   1:  PR[91,1] = PR[90,1] + 40.590;
   1:  PR[91,2] = PR[90,2] + 10.194;
   1:L PR[91] R[100]mm/sec CNT100;
   1:  PR[91,1] = PR[90,1] + 38.016;
   1:  PR[91,2] = PR[90,2] + 13.467;
   1:L PR[91] R[100]mm/sec CNT100;
   1:  PR[91,1] = PR[90,1] + 37.291;
   1:  PR[91,2] = PR[90,2] + 14.026;
   1:L PR[91] R[100]mm/sec CNT100;
   1:  PR[91,1] = PR[90,1] + 33.908;
   1:  PR[91,2] = PR[90,2] + 16.575;
   1:L PR[91] R[100]mm/sec CNT100;
   1:  PR[91,1] = PR[90,1] + 29.117;
   1:  PR[91,2] = PR[90,2] + 18.537;
   1:L PR[91] R[100]mm/sec CNT100;
   1:  PR[91,1] = PR[90,1] + 28.399;
   1:  PR[91,2] = PR[90,2] + 18.634;
   1:L PR[91] R[100]mm/sec CNT100;
   1:  PR[91,1] = PR[90,1] + 23.987;
   1:  PR[91,2] = PR[90,2] + 19.202;
   1:L PR[91] R[100]mm/sec CNT100;
   1:  PR[91,1] = PR[90,1] + 18.842;
   1:  PR[91,2] = PR[90,2] + 18.522;
   1:L PR[91] R[100]mm/sec CNT100;
   1:  PR[91,1] = PR[90,1] + 14.039;
   1:  PR[91,2] = PR[90,2] + 16.538;
   1:L PR[91] R[100]mm/sec CNT100;
   1:  PR[91,1] = PR[90,1] + 9.906;
   1:  PR[91,2] = PR[90,2] + 13.378;
   1:L PR[91] R[100]mm/sec CNT100;
   1:  PR[91,1] = PR[90,1] + 6.730;
   1:  PR[91,2] = PR[90,2] + 9.250;
   1:L PR[91] R[100]mm/sec CNT100;
   1:  PR[91,1] = PR[90,1] + 4.730;
   1:  PR[91,2] = PR[90,2] + 4.439;
   1:L PR[91] R[100]mm/sec CNT100;
   1:  PR[91,1] = PR[90,1] + 4.049;
   1:  PR[91,2] = PR[90,2] + -0.729;
   1:L PR[91] R[100]mm/sec CNT100;
   1:  PR[91,1] = PR[90,1] + 4.732;
   1:  PR[91,2] = PR[90,2] + -5.902;
   1:L PR[91] R[100]mm/sec CNT100;
   1:  PR[91,1] = PR[90,1] + 6.735;
   1:  PR[91,2] = PR[90,2] + -10.718;
   1:L PR[91] R[100]mm/sec CNT100;
   1:  PR[91,1] = PR[90,1] + 9.916;
   1:  PR[91,2] = PR[90,2] + -14.847;
   1:L PR[91] R[100]mm/sec CNT100;
   1:  PR[91,1] = PR[90,1] + 14.056;
   1:  PR[91,2] = PR[90,2] + -18.006;
   1:L PR[91] R[100]mm/sec CNT100;
   1:  PR[91,1] = PR[90,1] + 18.865;
   1:  PR[91,2] = PR[90,2] + -19.987;
   1:L PR[91] R[100]mm/sec CNT100;
   1:  PR[91,1] = PR[90,1] + 24.014;
   1:  PR[91,2] = PR[90,2] + -20.661;
   1:L PR[91] R[100]mm/sec CNT100;
   1:  PR[91,1] = PR[90,1] + 28.429;
   1:  PR[91,2] = PR[90,2] + -20.085;
   1:L PR[91] R[100]mm/sec CNT100;
   1:  PR[91,1] = PR[90,1] + 29.148;
   1:  PR[91,2] = PR[90,2] + -19.987;
   1:L PR[91] R[100]mm/sec CNT100;
   1:  PR[91,1] = PR[90,1] + 33.936;
   1:  PR[91,2] = PR[90,2] + -18.017;
   1:L PR[91] R[100]mm/sec CNT100;
   1:  PR[91,1] = PR[90,1] + 38.048;
   1:  PR[91,2] = PR[90,2] + -14.892;
   1:L PR[91] R[100]mm/sec CNT100;
   1:  PR[91,1] = PR[90,1] + 40.630;
   1:  PR[91,2] = PR[90,2] + -11.589;
   1:L PR[91] R[100]mm/sec CNT100;
   1:  PR[91,1] = PR[90,1] + 41.273;
   1:  PR[91,2] = PR[90,2] + -10.747;
   1:L PR[91] R[100]mm/sec CNT100;
   1:  PR[91,1] = PR[90,1] + 41.543;
   1:  PR[91,2] = PR[90,2] + -10.255;
   1:L PR[91] R[100]mm/sec CNT100;
   1:  PR[91,1] = PR[90,1] + 41.867;
   1:  PR[91,2] = PR[90,2] + -9.470;
   1:L PR[91] R[100]mm/sec CNT100;
   1:  PR[91,1] = PR[90,1] + 44.364;
   1:  PR[91,2] = PR[90,2] + -3.909;
   1:L PR[91] R[100]mm/sec CNT100;
   1:  PR[91,1] = PR[90,1] + 47.704;
   1:  PR[91,2] = PR[90,2] + -10.331;
   1:L PR[91] R[100]mm/sec CNT100;
   1:  PR[91,1] = PR[90,1] + 48.926;
   1:  PR[91,2] = PR[90,2] + -11.795;
   1:L PR[91] R[100]mm/sec CNT100;
   1:  PR[91,1] = PR[90,1] + 51.775;
   1:  PR[91,2] = PR[90,2] + -14.772;
   1:L PR[91] R[100]mm/sec CNT100;
   1:  PR[91,1] = PR[90,1] + 52.056;
   1:  PR[91,2] = PR[90,2] + -14.978;
   1:L PR[91] R[100]mm/sec CNT100;
   1:  PR[91,1] = PR[90,1] + 53.337;
   1:  PR[91,2] = PR[90,2] + -15.767;
   1:L PR[91] R[100]mm/sec CNT100;
   1:  PR[91,1] = PR[90,1] + 56.402;
   1:  PR[91,2] = PR[90,2] + -17.898;
   1:L PR[91] R[100]mm/sec CNT100;
   1:  PR[91,1] = PR[90,1] + 57.333;
   1:  PR[91,2] = PR[90,2] + -18.350;
   1:L PR[91] R[100]mm/sec CNT100;
   1:  PR[91,1] = PR[90,1] + 60.886;
   1:  PR[91,2] = PR[90,2] + -19.737;
   1:L PR[91] R[100]mm/sec CNT100;
   1:  PR[91,1] = PR[90,1] + 63.586;
   1:  PR[91,2] = PR[90,2] + -20.396;
   1:L PR[91] R[100]mm/sec CNT100;
   1:  PR[91,1] = PR[90,1] + 65.452;
   1:  PR[91,2] = PR[90,2] + -20.674;
   1:L PR[91] R[100]mm/sec CNT100;
   1:  PR[91,1] = PR[90,1] + 69.656;
   1:  PR[91,2] = PR[90,2] + -20.825;
   1:L PR[91] R[100]mm/sec CNT100;
   1:  PR[91,1] = PR[90,1] + 69.952;
   1:  PR[91,2] = PR[90,2] + -20.804;
   1:L PR[91] R[100]mm/sec CNT100;
   1:  PR[91,1] = PR[90,1] + 71.659;
   1:  PR[91,2] = PR[90,2] + -20.520;
   1:L PR[91] R[100]mm/sec CNT100;
   1:  PR[91,1] = PR[90,1] + 74.623;
   1:  PR[91,2] = PR[90,2] + -20.055;
   1:L PR[91] R[100]mm/sec CNT100;
   1:  PR[91,1] = PR[90,1] + 75.033;
   1:  PR[91,2] = PR[90,2] + -19.903;
   1:L PR[91] R[100]mm/sec CNT100;
   1:  PR[91,1] = PR[90,1] + 78.943;
   1:  PR[91,2] = PR[90,2] + -18.404;
   1:L PR[91] R[100]mm/sec CNT100;
   1:  PR[91,1] = PR[90,1] + 80.020;
   1:  PR[91,2] = PR[90,2] + -17.717;
   1:L PR[91] R[100]mm/sec CNT100;
   1:  PR[91,1] = PR[90,1] + 82.749;
   1:  PR[91,2] = PR[90,2] + -15.933;
   1:L PR[91] R[100]mm/sec CNT100;
   1:  PR[91,1] = PR[90,1] + 84.089;
   1:  PR[91,2] = PR[90,2] + -14.597;
   1:L PR[91] R[100]mm/sec CNT100;
   1:  PR[91,1] = PR[90,1] + 85.881;
   1:  PR[91,2] = PR[90,2] + -12.773;
   1:L PR[91] R[100]mm/sec CNT100;
   1:  PR[91,1] = PR[90,1] + 88.217;
   1:  PR[91,2] = PR[90,2] + -9.066;
   1:L PR[91] R[100]mm/sec CNT100;
   1:  PR[91,1] = PR[90,1] + 89.654;
   1:  PR[91,2] = PR[90,2] + -4.990;
   1:L PR[91] R[100]mm/sec CNT100;
   1:  PR[91,1] = PR[90,1] + 90.143;
   1:  PR[91,2] = PR[90,2] + -0.729;
   1:L PR[91] R[100]mm/sec CNT100;
   1:  PR[91,1] = PR[90,1] + 89.654;
   1:  PR[91,2] = PR[90,2] + 3.531;
   1:L PR[91] R[100]mm/sec CNT100;
   1:  PR[91,1] = PR[90,1] + 88.218;
   1:  PR[91,2] = PR[90,2] + 7.603;
   1:L PR[91] R[100]mm/sec CNT100;
   1:  PR[91,1] = PR[90,1] + 86.960;
   1:  PR[91,2] = PR[90,2] + 9.583;
   1:L PR[91] R[100]mm/sec CNT100;
   1:  PR[91,1] = PR[90,1] + 85.883;
   1:  PR[91,2] = PR[90,2] + 11.309;
   1:L PR[91] R[100]mm/sec CNT100;
   1:  PR[91,1] = PR[90,1] + 84.452;
   1:  PR[91,2] = PR[90,2] + 12.734;
   1:L PR[91] R[100]mm/sec CNT100;
   1:  PR[91,1] = PR[90,1] + 82.749;
   1:  PR[91,2] = PR[90,2] + 14.471;
   1:L PR[91] R[100]mm/sec CNT100;
   1:  PR[91,1] = PR[90,1] + 81.417;
   1:  PR[91,2] = PR[90,2] + 15.317;
   1:L PR[91] R[100]mm/sec CNT100;
   1:  PR[91,1] = PR[90,1] + 78.943;
   1:  PR[91,2] = PR[90,2] + 16.942;
   1:L PR[91] R[100]mm/sec CNT100;
   1:  PR[91,1] = PR[90,1] + 77.998;
   1:  PR[91,2] = PR[90,2] + 17.288;
   1:L PR[91] R[100]mm/sec CNT100;
   1:  PR[91,1] = PR[90,1] + 74.607;
   1:  PR[91,2] = PR[90,2] + 18.598;
   1:L PR[91] R[100]mm/sec CNT100;
   1:  PR[91,1] = PR[90,1] + 71.659;
   1:  PR[91,2] = PR[90,2] + 19.061;
   1:L PR[91] R[100]mm/sec CNT100;
   1:  PR[91,1] = PR[90,1] + 69.952;
   1:  PR[91,2] = PR[90,2] + 19.345;
   1:L PR[91] R[100]mm/sec CNT100TB   .50sec,CALL END_PUD;
   1:  PR[92] = PR[91];
   1:  PR[92,3] = PR[92,3] + 20;
   1:J PR[92] 10% FINE;
   1:  PR[91,1] = PR[90,1] + -21.225;
   1:  PR[91,2] = PR[90,2] + -20.035;
   1:  PR[92] = PR[91];
   1:  PR[92,3] = PR[92,3] + 20;
   1:J PR[92] 10% FINE;
   1:L PR[91] R[100]mm/sec CNT100;
   1:  CALL LASER_DRAHT_START;
   1:  PR[91,1] = PR[90,1] + -17.834;
   1:  PR[91,2] = PR[90,2] + -19.755;
   1:L PR[91] R[100]mm/sec CNT100;
   1:  PR[91,1] = PR[90,1] + -16.393;
   1:  PR[91,2] = PR[90,2] + -19.403;
   1:L PR[91] R[100]mm/sec CNT100;
   1:  PR[91,1] = PR[90,1] + -13.614;
   1:  PR[91,2] = PR[90,2] + -18.541;
   1:L PR[91] R[100]mm/sec CNT100;
   1:  PR[91,1] = PR[90,1] + -11.836;
   1:  PR[91,2] = PR[90,2] + -17.662;
   1:L PR[91] R[100]mm/sec CNT100;
   1:  PR[91,1] = PR[90,1] + -9.749;
   1:  PR[91,2] = PR[90,2] + -16.459;
   1:L PR[91] R[100]mm/sec CNT100;
   1:  PR[91,1] = PR[90,1] + -7.849;
   1:  PR[91,2] = PR[90,2] + -14.914;
   1:L PR[91] R[100]mm/sec CNT100;
   1:  PR[91,1] = PR[90,1] + -6.429;
   1:  PR[91,2] = PR[90,2] + -13.596;
   1:L PR[91] R[100]mm/sec CNT100;
   1:  PR[91,1] = PR[90,1] + -4.688;
   1:  PR[91,2] = PR[90,2] + -11.349;
   1:L PR[91] R[100]mm/sec CNT100;
   1:  PR[91,1] = PR[90,1] + -3.827;
   1:  PR[91,2] = PR[90,2] + -10.067;
   1:L PR[91] R[100]mm/sec CNT100;
   1:  PR[91,1] = PR[90,1] + -2.535;
   1:  PR[91,2] = PR[90,2] + -7.218;
   1:L PR[91] R[100]mm/sec CNT100;
   1:  PR[91,1] = PR[90,1] + -2.094;
   1:  PR[91,2] = PR[90,2] + -6.035;
   1:L PR[91] R[100]mm/sec CNT100;
   1:  PR[91,1] = PR[90,1] + -1.483;
   1:  PR[91,2] = PR[90,2] + -2.786;
   1:L PR[91] R[100]mm/sec CNT100;
   1:  PR[91,1] = PR[90,1] + -1.346;
   1:  PR[91,2] = PR[90,2] + -1.651;
   1:L PR[91] R[100]mm/sec CNT100;
   1:  PR[91,1] = PR[90,1] + -1.323;
   1:  PR[91,2] = PR[90,2] + -0.821;
   1:L PR[91] R[100]mm/sec CNT100;
   1:  PR[91,1] = PR[90,1] + -1.464;
   1:  PR[91,2] = PR[90,2] + 0.357;
   1:L PR[91] R[100]mm/sec CNT100;
   1:  PR[91,1] = PR[90,1] + -1.499;
   1:  PR[91,2] = PR[90,2] + 1.403;
   1:L PR[91] R[100]mm/sec CNT100;
   1:  PR[91,1] = PR[90,1] + -2.091;
   1:  PR[91,2] = PR[90,2] + 4.565;
   1:L PR[91] R[100]mm/sec CNT100;
   1:  PR[91,1] = PR[90,1] + -2.532;
   1:  PR[91,2] = PR[90,2] + 5.748;
   1:L PR[91] R[100]mm/sec CNT100;
   1:  PR[91,1] = PR[90,1] + -3.821;
   1:  PR[91,2] = PR[90,2] + 8.599;
   1:L PR[91] R[100]mm/sec CNT100;
   1:  PR[91,1] = PR[90,1] + -4.683;
   1:  PR[91,2] = PR[90,2] + 9.880;
   1:L PR[91] R[100]mm/sec CNT100;
   1:  PR[91,1] = PR[90,1] + -6.422;
   1:  PR[91,2] = PR[90,2] + 12.130;
   1:L PR[91] R[100]mm/sec CNT100;
   1:  PR[91,1] = PR[90,1] + -7.842;
   1:  PR[91,2] = PR[90,2] + 13.448;
   1:L PR[91] R[100]mm/sec CNT100;
   1:  PR[91,1] = PR[90,1] + -9.742;
   1:  PR[91,2] = PR[90,2] + 14.996;
   1:L PR[91] R[100]mm/sec CNT100;
   1:  PR[91,1] = PR[90,1] + -11.830;
   1:  PR[91,2] = PR[90,2] + 16.199;
   1:L PR[91] R[100]mm/sec CNT100;
   1:  PR[91,1] = PR[90,1] + -13.608;
   1:  PR[91,2] = PR[90,2] + 17.080;
   1:L PR[91] R[100]mm/sec CNT100;
   1:  PR[91,1] = PR[90,1] + -16.388;
   1:  PR[91,2] = PR[90,2] + 17.942;
   1:L PR[91] R[100]mm/sec CNT100;
   1:  PR[91,1] = PR[90,1] + -17.830;
   1:  PR[91,2] = PR[90,2] + 18.295;
   1:L PR[91] R[100]mm/sec CNT100;
   1:  PR[91,1] = PR[90,1] + -21.221;
   1:  PR[91,2] = PR[90,2] + 18.576;
   1:L PR[91] R[100]mm/sec CNT100;
   1:  PR[91,1] = PR[90,1] + -22.208;
   1:  PR[91,2] = PR[90,2] + 18.600;
   1:L PR[91] R[100]mm/sec CNT100;
   1:  PR[91,1] = PR[90,1] + -26.020;
   1:  PR[91,2] = PR[90,2] + 18.084;
   1:L PR[91] R[100]mm/sec CNT100;
   1:  PR[91,1] = PR[90,1] + -26.539;
   1:  PR[91,2] = PR[90,2] + 17.984;
   1:L PR[91] R[100]mm/sec CNT100;
   1:  PR[91,1] = PR[90,1] + -30.506;
   1:  PR[91,2] = PR[90,2] + 16.533;
   1:L PR[91] R[100]mm/sec CNT100;
   1:  PR[91,1] = PR[90,1] + -30.622;
   1:  PR[91,2] = PR[90,2] + 16.484;
   1:L PR[91] R[100]mm/sec CNT100;
   1:  PR[91,1] = PR[90,1] + -34.299;
   1:  PR[91,2] = PR[90,2] + 14.135;
   1:L PR[91] R[100]mm/sec CNT100;
   1:  PR[91,1] = PR[90,1] + -37.304;
   1:  PR[91,2] = PR[90,2] + 11.094;
   1:L PR[91] R[100]mm/sec CNT100;
   1:  PR[91,1] = PR[90,1] + -39.555;
   1:  PR[91,2] = PR[90,2] + 7.482;
   1:L PR[91] R[100]mm/sec CNT100;
   1:  PR[91,1] = PR[90,1] + -40.947;
   1:  PR[91,2] = PR[90,2] + 3.475;
   1:L PR[91] R[100]mm/sec CNT100;
   1:  PR[91,1] = PR[90,1] + -41.422;
   1:  PR[91,2] = PR[90,2] + -0.718;
   1:L PR[91] R[100]mm/sec CNT100;
   1:  PR[91,1] = PR[90,1] + -41.389;
   1:  PR[91,2] = PR[90,2] + -0.982;
   1:L PR[91] R[100]mm/sec CNT100;
   1:  PR[91,1] = PR[90,1] + -40.947;
   1:  PR[91,2] = PR[90,2] + -4.935;
   1:L PR[91] R[100]mm/sec CNT100;
   1:  PR[91,1] = PR[90,1] + -39.555;
   1:  PR[91,2] = PR[90,2] + -8.940;
   1:L PR[91] R[100]mm/sec CNT100;
   1:  PR[91,1] = PR[90,1] + -37.304;
   1:  PR[91,2] = PR[90,2] + -12.552;
   1:L PR[91] R[100]mm/sec CNT100;
   1:  PR[91,1] = PR[90,1] + -34.300;
   1:  PR[91,2] = PR[90,2] + -15.594;
   1:L PR[91] R[100]mm/sec CNT100;
   1:  PR[91,1] = PR[90,1] + -30.622;
   1:  PR[91,2] = PR[90,2] + -17.943;
   1:L PR[91] R[100]mm/sec CNT100;
   1:  PR[91,1] = PR[90,1] + -30.507;
   1:  PR[91,2] = PR[90,2] + -17.992;
   1:L PR[91] R[100]mm/sec CNT100;
   1:  PR[91,1] = PR[90,1] + -26.540;
   1:  PR[91,2] = PR[90,2] + -19.442;
   1:L PR[91] R[100]mm/sec CNT100;
   1:  PR[91,1] = PR[90,1] + -26.022;
   1:  PR[91,2] = PR[90,2] + -19.543;
   1:L PR[91] R[100]mm/sec CNT100;
   1:  PR[91,1] = PR[90,1] + -22.211;
   1:  PR[91,2] = PR[90,2] + -20.059;
   1:L PR[91] R[100]mm/sec CNT100;
   1:  PR[91,1] = PR[90,1] + -21.225;
   1:  PR[91,2] = PR[90,2] + -20.035;
   1:L PR[91] R[100]mm/sec CNT100TB   .50sec,CALL END_PUD;
   1:  PR[92] = PR[91];
   1:  PR[92,3] = PR[92,3] + 20;
   1:J PR[92] 10% FINE;
   1:  PR[91,1] = PR[90,1] + -89.612;
   1:  PR[91,2] = PR[90,2] + -4.603;
   1:  PR[92] = PR[91];
   1:  PR[92,3] = PR[92,3] + 20;
   1:J PR[92] 10% FINE;
   1:L PR[91] R[100]mm/sec CNT100;
   1:  CALL LASER_DRAHT_START;
   1:  PR[91,1] = PR[90,1] + -88.374;
   1:  PR[91,2] = PR[90,2] + -8.320;
   1:L PR[91] R[100]mm/sec CNT100;
   1:  PR[91,1] = PR[90,1] + -86.359;
   1:  PR[91,2] = PR[90,2] + -11.734;
   1:L PR[91] R[100]mm/sec CNT100;
   1:  PR[91,1] = PR[90,1] + -83.646;
   1:  PR[91,2] = PR[90,2] + -14.700;
   1:L PR[91] R[100]mm/sec CNT100;
   1:  PR[91,1] = PR[90,1] + -81.589;
   1:  PR[91,2] = PR[90,2] + -16.174;
   1:L PR[91] R[100]mm/sec CNT100;
   1:  PR[91,1] = PR[90,1] + -80.327;
   1:  PR[91,2] = PR[90,2] + -17.098;
   1:L PR[91] R[100]mm/sec CNT100;
   1:  PR[91,1] = PR[90,1] + -78.378;
   1:  PR[91,2] = PR[90,2] + -17.969;
   1:L PR[91] R[100]mm/sec CNT100;
   1:  PR[91,1] = PR[90,1] + -76.545;
   1:  PR[91,2] = PR[90,2] + -18.813;
   1:L PR[91] R[100]mm/sec CNT100;
   1:  PR[91,1] = PR[90,1] + -74.930;
   1:  PR[91,2] = PR[90,2] + -19.175;
   1:L PR[91] R[100]mm/sec CNT100;
   1:  PR[91,1] = PR[90,1] + -72.446;
   1:  PR[91,2] = PR[90,2] + -19.767;
   1:L PR[91] R[100]mm/sec CNT100;
   1:  PR[91,1] = PR[90,1] + -71.357;
   1:  PR[91,2] = PR[90,2] + -19.791;
   1:L PR[91] R[100]mm/sec CNT100;
   1:  PR[91,1] = PR[90,1] + -68.183;
   1:  PR[91,2] = PR[90,2] + -19.907;
   1:L PR[91] R[100]mm/sec CNT100;
   1:  PR[91,1] = PR[90,1] + -63.917;
   1:  PR[91,2] = PR[90,2] + -19.209;
   1:L PR[91] R[100]mm/sec CNT100;
   1:  PR[91,1] = PR[90,1] + -60.270;
   1:  PR[91,2] = PR[90,2] + -17.914;
   1:L PR[91] R[100]mm/sec CNT100;
   1:  PR[91,1] = PR[90,1] + -59.627;
   1:  PR[91,2] = PR[90,2] + -17.699;
   1:L PR[91] R[100]mm/sec CNT100;
   1:  PR[91,1] = PR[90,1] + -57.061;
   1:  PR[91,2] = PR[90,2] + -16.158;
   1:L PR[91] R[100]mm/sec CNT100;
   1:  PR[91,1] = PR[90,1] + -55.776;
   1:  PR[91,2] = PR[90,2] + -15.417;
   1:L PR[91] R[100]mm/sec CNT100;
   1:  PR[91,1] = PR[90,1] + -54.204;
   1:  PR[91,2] = PR[90,2] + -13.950;
   1:L PR[91] R[100]mm/sec CNT100;
   1:  PR[91,1] = PR[90,1] + -52.527;
   1:  PR[91,2] = PR[90,2] + -12.434;
   1:L PR[91] R[100]mm/sec CNT100;
   1:  PR[91,1] = PR[90,1] + -51.753;
   1:  PR[91,2] = PR[90,2] + -11.300;
   1:L PR[91] R[100]mm/sec CNT100;
   1:  PR[91,1] = PR[90,1] + -50.050;
   1:  PR[91,2] = PR[90,2] + -8.871;
   1:L PR[91] R[100]mm/sec CNT100;
   1:  PR[91,1] = PR[90,1] + -48.508;
   1:  PR[91,2] = PR[90,2] + -4.909;
   1:L PR[91] R[100]mm/sec CNT100;
   1:  PR[91,1] = PR[90,1] + -48.480;
   1:  PR[91,2] = PR[90,2] + -4.681;
   1:L PR[91] R[100]mm/sec CNT100;
   1:  PR[91,1] = PR[90,1] + -48.428;
   1:  PR[91,2] = PR[90,2] + -3.939;
   1:L PR[91] R[100]mm/sec CNT100;
   1:  PR[91,1] = PR[90,1] + -48.016;
   1:  PR[91,2] = PR[90,2] + -0.731;
   1:L PR[91] R[100]mm/sec CNT100;
   1:  PR[91,1] = PR[90,1] + -48.104;
   1:  PR[91,2] = PR[90,2] + -0.048;
   1:L PR[91] R[100]mm/sec CNT100;
   1:  PR[91,1] = PR[90,1] + -48.291;
   1:  PR[91,2] = PR[90,2] + 2.128;
   1:L PR[91] R[100]mm/sec CNT100;
   1:  PR[91,1] = PR[90,1] + -48.464;
   1:  PR[91,2] = PR[90,2] + 3.428;
   1:L PR[91] R[100]mm/sec CNT100;
   1:  PR[91,1] = PR[90,1] + -50.071;
   1:  PR[91,2] = PR[90,2] + 7.381;
   1:L PR[91] R[100]mm/sec CNT100;
   1:  PR[91,1] = PR[90,1] + -52.667;
   1:  PR[91,2] = PR[90,2] + 10.955;
   1:L PR[91] R[100]mm/sec CNT100;
   1:  PR[91,1] = PR[90,1] + -55.865;
   1:  PR[91,2] = PR[90,2] + 13.968;
   1:L PR[91] R[100]mm/sec CNT100;
   1:  PR[91,1] = PR[90,1] + -59.639;
   1:  PR[91,2] = PR[90,2] + 16.261;
   1:L PR[91] R[100]mm/sec CNT100;
   1:  PR[91,1] = PR[90,1] + -61.792;
   1:  PR[91,2] = PR[90,2] + 17.051;
   1:L PR[91] R[100]mm/sec CNT100;
   1:  PR[91,1] = PR[90,1] + -63.801;
   1:  PR[91,2] = PR[90,2] + 17.766;
   1:L PR[91] R[100]mm/sec CNT100;
   1:  PR[91,1] = PR[90,1] + -68.191;
   1:  PR[91,2] = PR[90,2] + 18.444;
   1:L PR[91] R[100]mm/sec CNT100;
   1:  PR[91,1] = PR[90,1] + -72.567;
   1:  PR[91,2] = PR[90,2] + 18.287;
   1:L PR[91] R[100]mm/sec CNT100;
   1:  PR[91,1] = PR[90,1] + -76.629;
   1:  PR[91,2] = PR[90,2] + 17.342;
   1:L PR[91] R[100]mm/sec CNT100;
   1:  PR[91,1] = PR[90,1] + -80.374;
   1:  PR[91,2] = PR[90,2] + 15.635;
   1:L PR[91] R[100]mm/sec CNT100;
   1:  PR[91,1] = PR[90,1] + -83.658;
   1:  PR[91,2] = PR[90,2] + 13.247;
   1:L PR[91] R[100]mm/sec CNT100;
   1:  PR[91,1] = PR[90,1] + -86.351;
   1:  PR[91,2] = PR[90,2] + 10.282;
   1:L PR[91] R[100]mm/sec CNT100;
   1:  PR[91,1] = PR[90,1] + -88.351;
   1:  PR[91,2] = PR[90,2] + 6.868;
   1:L PR[91] R[100]mm/sec CNT100;
   1:  PR[91,1] = PR[90,1] + -89.581;
   1:  PR[91,2] = PR[90,2] + 3.146;
   1:L PR[91] R[100]mm/sec CNT100;
   1:  PR[91,1] = PR[90,1] + -89.835;
   1:  PR[91,2] = PR[90,2] + 0.801;
   1:L PR[91] R[100]mm/sec CNT100;
   1:  PR[91,1] = PR[90,1] + -89.986;
   1:  PR[91,2] = PR[90,2] + 0.050;
   1:L PR[91] R[100]mm/sec CNT100;
   1:  PR[91,1] = PR[90,1] + -90.069;
   1:  PR[91,2] = PR[90,2] + -0.728;
   1:L PR[91] R[100]mm/sec CNT100;
   1:  PR[91,1] = PR[90,1] + -89.760;
   1:  PR[91,2] = PR[90,2] + -3.570;
   1:L PR[91] R[100]mm/sec CNT100;
   1:  PR[91,1] = PR[90,1] + -89.687;
   1:  PR[91,2] = PR[90,2] + -3.899;
   1:L PR[91] R[100]mm/sec CNT100;
   1:  PR[91,1] = PR[90,1] + -89.612;
   1:  PR[91,2] = PR[90,2] + -4.603;
   1:L PR[91] R[100]mm/sec CNT100TB   .50sec,CALL END_PUD;
   1:  PR[92] = PR[91];
   1:  PR[92,3] = PR[92,3] + 20;
   1:J PR[92] 10% FINE;
   1:  PR[91] = PR[90];
   1:  PR[91,1] = PR[90,1] + 48.448;
   1:  PR[91,2] = PR[90,2] + -12.683;
   1:  PR[91,3] = PR[90,3] + 36.595;
   1:  PR[92] = PR[91];
   1:  PR[92,3] = PR[92,3] + 20;
   1:J PR[92] 10% FINE;
   1:L PR[91] R[100]mm/sec CNT100;
   1:  CALL LASER_DRAHT_START;
   1:  PR[91,1] = PR[90,1] + 50.330;
   1:  PR[91,2] = PR[90,2] + -14.650;
   1:L PR[91] R[100]mm/sec CNT100;
   1:  PR[91,1] = PR[90,1] + 51.696;
   1:  PR[91,2] = PR[90,2] + -15.650;
   1:L PR[91] R[100]mm/sec CNT100;
   1:  PR[91,1] = PR[90,1] + 55.883;
   1:  PR[91,2] = PR[90,2] + -18.236;
   1:L PR[91] R[100]mm/sec CNT100;
   1:  PR[91,1] = PR[90,1] + 60.564;
   1:  PR[91,2] = PR[90,2] + -20.064;
   1:L PR[91] R[100]mm/sec CNT100;
   1:  PR[91,1] = PR[90,1] + 62.228;
   1:  PR[91,2] = PR[90,2] + -20.470;
   1:L PR[91] R[100]mm/sec CNT100;
   1:  PR[91,1] = PR[90,1] + 65.235;
   1:  PR[91,2] = PR[90,2] + -20.918;
   1:L PR[91] R[100]mm/sec CNT100;
   1:  PR[91,1] = PR[90,1] + 68.507;
   1:  PR[91,2] = PR[90,2] + -21.035;
   1:L PR[91] R[100]mm/sec CNT100;
   1:  PR[91,1] = PR[90,1] + 69.807;
   1:  PR[91,2] = PR[90,2] + -20.945;
   1:L PR[91] R[100]mm/sec CNT100;
   1:  PR[91,1] = PR[90,1] + 74.194;
   1:  PR[91,2] = PR[90,2] + -20.214;
   1:L PR[91] R[100]mm/sec CNT100;
   1:  PR[91,1] = PR[90,1] + 78.605;
   1:  PR[91,2] = PR[90,2] + -18.523;
   1:L PR[91] R[100]mm/sec CNT100;
   1:  PR[91,1] = PR[90,1] + 79.073;
   1:  PR[91,2] = PR[90,2] + -18.225;
   1:L PR[91] R[100]mm/sec CNT100;
   1:  PR[91,1] = PR[90,1] + 82.426;
   1:  PR[91,2] = PR[90,2] + -16.033;
   1:L PR[91] R[100]mm/sec CNT100;
   1:  PR[91,1] = PR[90,1] + 85.579;
   1:  PR[91,2] = PR[90,2] + -12.844;
   1:L PR[91] R[100]mm/sec CNT100;
   1:  PR[91,1] = PR[90,1] + 87.923;
   1:  PR[91,2] = PR[90,2] + -9.115;
   1:L PR[91] R[100]mm/sec CNT100;
   1:  PR[91,1] = PR[90,1] + 89.365;
   1:  PR[91,2] = PR[90,2] + -5.015;
   1:L PR[91] R[100]mm/sec CNT100;
   1:  PR[91,1] = PR[90,1] + 89.856;
   1:  PR[91,2] = PR[90,2] + -0.729;
   1:L PR[91] R[100]mm/sec CNT100;
   1:  PR[91,1] = PR[90,1] + 89.365;
   1:  PR[91,2] = PR[90,2] + 3.556;
   1:L PR[91] R[100]mm/sec CNT100;
   1:  PR[91,1] = PR[90,1] + 87.924;
   1:  PR[91,2] = PR[90,2] + 7.651;
   1:L PR[91] R[100]mm/sec CNT100;
   1:  PR[91,1] = PR[90,1] + 86.953;
   1:  PR[91,2] = PR[90,2] + 9.179;
   1:L PR[91] R[100]mm/sec CNT100;
   1:  PR[91,1] = PR[90,1] + 85.580;
   1:  PR[91,2] = PR[90,2] + 11.381;
   1:L PR[91] R[100]mm/sec CNT100;
   1:  PR[91,1] = PR[90,1] + 84.536;
   1:  PR[91,2] = PR[90,2] + 12.421;
   1:L PR[91] R[100]mm/sec CNT100;
   1:  PR[91,1] = PR[90,1] + 82.432;
   1:  PR[91,2] = PR[90,2] + 14.567;
   1:L PR[91] R[100]mm/sec CNT100;
   1:  PR[91,1] = PR[90,1] + 81.577;
   1:  PR[91,2] = PR[90,2] + 15.110;
   1:L PR[91] R[100]mm/sec CNT100;
   1:  PR[91,1] = PR[90,1] + 78.593;
   1:  PR[91,2] = PR[90,2] + 17.069;
   1:L PR[91] R[100]mm/sec CNT100;
   1:  PR[91,1] = PR[90,1] + 74.194;
   1:  PR[91,2] = PR[90,2] + 18.755;
   1:L PR[91] R[100]mm/sec CNT100;
   1:  PR[91,1] = PR[90,1] + 69.807;
   1:  PR[91,2] = PR[90,2] + 19.486;
   1:L PR[91] R[100]mm/sec CNT100;
   1:  PR[91,1] = PR[90,1] + 68.508;
   1:  PR[91,2] = PR[90,2] + 19.576;
   1:L PR[91] R[100]mm/sec CNT100;
   1:  PR[91,1] = PR[90,1] + 65.236;
   1:  PR[91,2] = PR[90,2] + 19.459;
   1:L PR[91] R[100]mm/sec CNT100;
   1:  PR[91,1] = PR[90,1] + 62.229;
   1:  PR[91,2] = PR[90,2] + 19.012;
   1:L PR[91] R[100]mm/sec CNT100;
   1:  PR[91,1] = PR[90,1] + 60.565;
   1:  PR[91,2] = PR[90,2] + 18.606;
   1:L PR[91] R[100]mm/sec CNT100;
   1:  PR[91,1] = PR[90,1] + 55.885;
   1:  PR[91,2] = PR[90,2] + 16.778;
   1:L PR[91] R[100]mm/sec CNT100;
   1:  PR[91,1] = PR[90,1] + 51.681;
   1:  PR[91,2] = PR[90,2] + 14.184;
   1:L PR[91] R[100]mm/sec CNT100;
   1:  PR[91,1] = PR[90,1] + 50.297;
   1:  PR[91,2] = PR[90,2] + 13.161;
   1:L PR[91] R[100]mm/sec CNT100;
   1:  PR[91,1] = PR[90,1] + 48.417;
   1:  PR[91,2] = PR[90,2] + 11.199;
   1:L PR[91] R[100]mm/sec CNT100;
   1:  PR[91,1] = PR[90,1] + 46.303;
   1:  PR[91,2] = PR[90,2] + 8.631;
   1:L PR[91] R[100]mm/sec CNT100;
   1:  PR[91,1] = PR[90,1] + 43.815;
   1:  PR[91,2] = PR[90,2] + 3.885;
   1:L PR[91] R[100]mm/sec CNT100;
   1:  PR[91,1] = PR[90,1] + 41.685;
   1:  PR[91,2] = PR[90,2] + 8.704;
   1:L PR[91] R[100]mm/sec CNT100;
   1:  PR[91,1] = PR[90,1] + 41.318;
   1:  PR[91,2] = PR[90,2] + 9.380;
   1:L PR[91] R[100]mm/sec CNT100;
   1:  PR[91,1] = PR[90,1] + 40.909;
   1:  PR[91,2] = PR[90,2] + 9.927;
   1:L PR[91] R[100]mm/sec CNT100;
   1:  PR[91,1] = PR[90,1] + 38.040;
   1:  PR[91,2] = PR[90,2] + 13.576;
   1:L PR[91] R[100]mm/sec CNT100;
   1:  PR[91,1] = PR[90,1] + 33.895;
   1:  PR[91,2] = PR[90,2] + 16.707;
   1:L PR[91] R[100]mm/sec CNT100;
   1:  PR[91,1] = PR[90,1] + 29.079;
   1:  PR[91,2] = PR[90,2] + 18.676;
   1:L PR[91] R[100]mm/sec CNT100;
   1:  PR[91,1] = PR[90,1] + 23.909;
   1:  PR[91,2] = PR[90,2] + 19.344;
   1:L PR[91] R[100]mm/sec CNT100;
   1:  PR[91,1] = PR[90,1] + 18.731;
   1:  PR[91,2] = PR[90,2] + 18.658;
   1:L PR[91] R[100]mm/sec CNT100;
   1:  PR[91,1] = PR[90,1] + 13.896;
   1:  PR[91,2] = PR[90,2] + 16.659;
   1:L PR[91] R[100]mm/sec CNT100;
   1:  PR[91,1] = PR[90,1] + 9.735;
   1:  PR[91,2] = PR[90,2] + 13.476;
   1:L PR[91] R[100]mm/sec CNT100;
   1:  PR[91,1] = PR[90,1] + 6.536;
   1:  PR[91,2] = PR[90,2] + 9.323;
   1:L PR[91] R[100]mm/sec CNT100;
   1:  PR[91,1] = PR[90,1] + 4.500;
   1:  PR[91,2] = PR[90,2] + 4.453;
   1:L PR[91] R[100]mm/sec CNT100;
   1:  PR[91,1] = PR[90,1] + 4.494;
   1:  PR[91,2] = PR[90,2] + 4.429;
   1:L PR[91] R[100]mm/sec CNT100;
   1:  PR[91,1] = PR[90,1] + 3.813;
   1:  PR[91,2] = PR[90,2] + -0.613;
   1:L PR[91] R[100]mm/sec CNT100;
   1:  PR[91,2] = PR[90,2] + -0.630;
   1:L PR[91] R[100]mm/sec CNT100;
   1:  PR[91,1] = PR[90,1] + 4.449;
   1:  PR[91,2] = PR[90,2] + -5.418;
   1:L PR[91] R[100]mm/sec CNT100;
   1:  PR[91,1] = PR[90,1] + 4.467;
   1:  PR[91,2] = PR[90,2] + -5.695;
   1:L PR[91] R[100]mm/sec CNT100;
   1:  PR[91,1] = PR[90,1] + 4.495;
   1:  PR[91,2] = PR[90,2] + -5.897;
   1:L PR[91] R[100]mm/sec CNT100;
   1:  PR[91,1] = PR[90,1] + 6.537;
   1:  PR[91,2] = PR[90,2] + -10.785;
   1:L PR[91] R[100]mm/sec CNT100;
   1:  PR[91,1] = PR[90,1] + 9.746;
   1:  PR[91,2] = PR[90,2] + -14.946;
   1:L PR[91] R[100]mm/sec CNT100;
   1:  PR[91,1] = PR[90,1] + 13.914;
   1:  PR[91,2] = PR[90,2] + -18.128;
   1:L PR[91] R[100]mm/sec CNT100;
   1:  PR[91,1] = PR[90,1] + 18.756;
   1:  PR[91,2] = PR[90,2] + -20.123;
   1:L PR[91] R[100]mm/sec CNT100;
   1:  PR[91,1] = PR[90,1] + 23.939;
   1:  PR[91,2] = PR[90,2] + -20.803;
   1:L PR[91] R[100]mm/sec CNT100;
   1:  PR[91,1] = PR[90,1] + 29.112;
   1:  PR[91,2] = PR[90,2] + -20.126;
   1:L PR[91] R[100]mm/sec CNT100;
   1:  PR[91,1] = PR[90,1] + 33.928;
   1:  PR[91,2] = PR[90,2] + -18.147;
   1:L PR[91] R[100]mm/sec CNT100;
   1:  PR[91,1] = PR[90,1] + 38.068;
   1:  PR[91,2] = PR[90,2] + -15.007;
   1:L PR[91] R[100]mm/sec CNT100;
   1:  PR[91,1] = PR[90,1] + 41.323;
   1:  PR[91,2] = PR[90,2] + -10.829;
   1:L PR[91] R[100]mm/sec CNT100;
   1:  PR[91,1] = PR[90,1] + 41.633;
   1:  PR[91,2] = PR[90,2] + -10.265;
   1:L PR[91] R[100]mm/sec CNT100;
   1:  PR[91,1] = PR[90,1] + 41.768;
   1:  PR[91,2] = PR[90,2] + -9.937;
   1:L PR[91] R[100]mm/sec CNT100;
   1:  PR[91,1] = PR[90,1] + 43.847;
   1:  PR[91,2] = PR[90,2] + -5.391;
   1:L PR[91] R[100]mm/sec CNT100;
   1:  PR[91,1] = PR[90,1] + 46.344;
   1:  PR[91,2] = PR[90,2] + -10.163;
   1:L PR[91] R[100]mm/sec CNT100;
   1:  PR[91,1] = PR[90,1] + 48.448;
   1:  PR[91,2] = PR[90,2] + -12.683;
   1:L PR[91] R[100]mm/sec CNT100TB   .50sec,CALL END_PUD;
   1:  PR[92] = PR[91];
   1:  PR[92,3] = PR[92,3] + 20;
   1:J PR[92] 10% FINE;
   1:  PR[91,1] = PR[90,1] + -9.454;
   1:  PR[91,2] = PR[90,2] + -16.672;
   1:  PR[92] = PR[91];
   1:  PR[92,3] = PR[92,3] + 20;
   1:J PR[92] 10% FINE;
   1:L PR[91] R[100]mm/sec CNT100;
   1:  CALL LASER_DRAHT_START;
   1:  PR[91,1] = PR[90,1] + -7.029;
   1:  PR[91,2] = PR[90,2] + -14.701;
   1:L PR[91] R[100]mm/sec CNT100;
   1:  PR[91,1] = PR[90,1] + -6.085;
   1:  PR[91,2] = PR[90,2] + -13.824;
   1:L PR[91] R[100]mm/sec CNT100;
   1:  PR[91,1] = PR[90,1] + -3.923;
   1:  PR[91,2] = PR[90,2] + -11.032;
   1:L PR[91] R[100]mm/sec CNT100;
   1:  PR[91,1] = PR[90,1] + -3.430;
   1:  PR[91,2] = PR[90,2] + -10.299;
   1:L PR[91] R[100]mm/sec CNT100;
   1:  PR[91,1] = PR[90,1] + -1.852;
   1:  PR[91,2] = PR[90,2] + -6.817;
   1:L PR[91] R[100]mm/sec CNT100;
   1:  PR[91,1] = PR[90,1] + -1.643;
   1:  PR[91,2] = PR[90,2] + -6.258;
   1:L PR[91] R[100]mm/sec CNT100;
   1:  PR[91,1] = PR[90,1] + -0.903;
   1:  PR[91,2] = PR[90,2] + -2.322;
   1:L PR[91] R[100]mm/sec CNT100;
   1:  PR[91,1] = PR[90,1] + -0.847;
   1:  PR[91,2] = PR[90,2] + -1.858;
   1:L PR[91] R[100]mm/sec CNT100;
   1:  PR[91,1] = PR[90,1] + -0.818;
   1:  PR[91,2] = PR[90,2] + -0.821;
   1:L PR[91] R[100]mm/sec CNT100;
   1:  PR[91,1] = PR[90,1] + -0.877;
   1:  PR[91,2] = PR[90,2] + -0.329;
   1:L PR[91] R[100]mm/sec CNT100;
   1:  PR[91,1] = PR[90,1] + -0.919;
   1:  PR[91,2] = PR[90,2] + 0.936;
   1:L PR[91] R[100]mm/sec CNT100;
   1:  PR[91,1] = PR[90,1] + -1.639;
   1:  PR[91,2] = PR[90,2] + 4.785;
   1:L PR[91] R[100]mm/sec CNT100;
   1:  PR[91,1] = PR[90,1] + -1.847;
   1:  PR[91,2] = PR[90,2] + 5.344;
   1:L PR[91] R[100]mm/sec CNT100;
   1:  PR[91,1] = PR[90,1] + -3.423;
   1:  PR[91,2] = PR[90,2] + 8.829;
   1:L PR[91] R[100]mm/sec CNT100;
   1:  PR[91,1] = PR[90,1] + -3.916;
   1:  PR[91,2] = PR[90,2] + 9.561;
   1:L PR[91] R[100]mm/sec CNT100;
   1:  PR[91,1] = PR[90,1] + -6.077;
   1:  PR[91,2] = PR[90,2] + 12.357;
   1:L PR[91] R[100]mm/sec CNT100;
   1:  PR[91,1] = PR[90,1] + -7.021;
   1:  PR[91,2] = PR[90,2] + 13.233;
   1:L PR[91] R[100]mm/sec CNT100;
   1:  PR[91,1] = PR[90,1] + -9.446;
   1:  PR[91,2] = PR[90,2] + 15.208;
   1:L PR[91] R[100]mm/sec CNT100;
   1:  PR[91,1] = PR[90,1] + -10.985;
   1:  PR[91,2] = PR[90,2] + 16.095;
   1:L PR[91] R[100]mm/sec CNT100;
   1:  PR[91,1] = PR[90,1] + -13.352;
   1:  PR[91,2] = PR[90,2] + 17.268;
   1:L PR[91] R[100]mm/sec CNT100;
   1:  PR[91,1] = PR[90,1] + -15.549;
   1:  PR[91,2] = PR[90,2] + 17.949;
   1:L PR[91] R[100]mm/sec CNT100;
   1:  PR[91,1] = PR[90,1] + -17.606;
   1:  PR[91,2] = PR[90,2] + 18.453;
   1:L PR[91] R[100]mm/sec CNT100;
   1:  PR[91,1] = PR[90,1] + -20.415;
   1:  PR[91,2] = PR[90,2] + 18.686;
   1:L PR[91] R[100]mm/sec CNT100;
   1:  PR[91,1] = PR[90,1] + -22.007;
   1:  PR[91,2] = PR[90,2] + 18.725;
   1:L PR[91] R[100]mm/sec CNT100;
   1:  PR[91,1] = PR[90,1] + -25.267;
   1:  PR[91,2] = PR[90,2] + 18.283;
   1:L PR[91] R[100]mm/sec CNT100;
   1:  PR[91,1] = PR[90,1] + -26.352;
   1:  PR[91,2] = PR[90,2] + 18.074;
   1:L PR[91] R[100]mm/sec CNT100;
   1:  PR[91,1] = PR[90,1] + -29.822;
   1:  PR[91,2] = PR[90,2] + 16.806;
   1:L PR[91] R[100]mm/sec CNT100;
   1:  PR[91,1] = PR[90,1] + -30.442;
   1:  PR[91,2] = PR[90,2] + 16.541;
   1:L PR[91] R[100]mm/sec CNT100;
   1:  PR[91,1] = PR[90,1] + -33.828;
   1:  PR[91,2] = PR[90,2] + 14.379;
   1:L PR[91] R[100]mm/sec CNT100;
   1:  PR[91,1] = PR[90,1] + -34.088;
   1:  PR[91,2] = PR[90,2] + 14.194;
   1:L PR[91] R[100]mm/sec CNT100;
   1:  PR[91,1] = PR[90,1] + -37.092;
   1:  PR[91,2] = PR[90,2] + 11.178;
   1:L PR[91] R[100]mm/sec CNT100;
   1:  PR[91,1] = PR[90,1] + -37.122;
   1:  PR[91,2] = PR[90,2] + 11.145;
   1:L PR[91] R[100]mm/sec CNT100;
   1:  PR[91,1] = PR[90,1] + -39.423;
   1:  PR[91,2] = PR[90,2] + 7.491;
   1:L PR[91] R[100]mm/sec CNT100;
   1:  PR[91,1] = PR[90,1] + -40.821;
   1:  PR[91,2] = PR[90,2] + 3.489;
   1:L PR[91] R[100]mm/sec CNT100;
   1:  PR[91,1] = PR[90,1] + -41.294;
   1:  PR[91,2] = PR[90,2] + -0.729;
   1:L PR[91] R[100]mm/sec CNT100;
   1:  PR[91,1] = PR[90,1] + -40.821;
   1:  PR[91,2] = PR[90,2] + -4.948;
   1:L PR[91] R[100]mm/sec CNT100;
   1:  PR[91,1] = PR[90,1] + -39.424;
   1:  PR[91,2] = PR[90,2] + -8.948;
   1:L PR[91] R[100]mm/sec CNT100;
   1:  PR[91,1] = PR[90,1] + -37.152;
   1:  PR[91,2] = PR[90,2] + -12.572;
   1:L PR[91] R[100]mm/sec CNT100;
   1:  PR[91,1] = PR[90,1] + -37.092;
   1:  PR[91,2] = PR[90,2] + -12.637;
   1:L PR[91] R[100]mm/sec CNT100;
   1:  PR[91,1] = PR[90,1] + -34.089;
   1:  PR[91,2] = PR[90,2] + -15.652;
   1:L PR[91] R[100]mm/sec CNT100;
   1:  PR[91,1] = PR[90,1] + -33.829;
   1:  PR[91,2] = PR[90,2] + -15.837;
   1:L PR[91] R[100]mm/sec CNT100;
   1:  PR[91,1] = PR[90,1] + -30.443;
   1:  PR[91,2] = PR[90,2] + -17.999;
   1:L PR[91] R[100]mm/sec CNT100;
   1:  PR[91,1] = PR[90,1] + -29.824;
   1:  PR[91,2] = PR[90,2] + -18.264;
   1:L PR[91] R[100]mm/sec CNT100;
   1:  PR[91,1] = PR[90,1] + -26.355;
   1:  PR[91,2] = PR[90,2] + -19.532;
   1:L PR[91] R[100]mm/sec CNT100;
   1:  PR[91,1] = PR[90,1] + -25.271;
   1:  PR[91,2] = PR[90,2] + -19.742;
   1:L PR[91] R[100]mm/sec CNT100;
   1:  PR[91,1] = PR[90,1] + -22.011;
   1:  PR[91,2] = PR[90,2] + -20.183;
   1:L PR[91] R[100]mm/sec CNT100;
   1:  PR[91,1] = PR[90,1] + -20.420;
   1:  PR[91,2] = PR[90,2] + -20.145;
   1:L PR[91] R[100]mm/sec CNT100;
   1:  PR[91,1] = PR[90,1] + -17.612;
   1:  PR[91,2] = PR[90,2] + -19.913;
   1:L PR[91] R[100]mm/sec CNT100;
   1:  PR[91,1] = PR[90,1] + -15.556;
   1:  PR[91,2] = PR[90,2] + -19.411;
   1:L PR[91] R[100]mm/sec CNT100;
   1:  PR[91,1] = PR[90,1] + -13.359;
   1:  PR[91,2] = PR[90,2] + -18.730;
   1:L PR[91] R[100]mm/sec CNT100;
   1:  PR[91,1] = PR[90,1] + -10.994;
   1:  PR[91,2] = PR[90,2] + -17.559;
   1:L PR[91] R[100]mm/sec CNT100;
   1:  PR[91,1] = PR[90,1] + -9.454;
   1:  PR[91,2] = PR[90,2] + -16.672;
   1:L PR[91] R[100]mm/sec CNT100TB   .50sec,CALL END_PUD;
   1:  PR[92] = PR[91];
   1:  PR[92,3] = PR[92,3] + 20;
   1:J PR[92] 10% FINE;
   1:  PR[91,1] = PR[90,1] + -88.029;
   1:  PR[91,2] = PR[90,2] + -8.350;
   1:  PR[92] = PR[91];
   1:  PR[92,3] = PR[92,3] + 20;
   1:J PR[92] 10% FINE;
   1:L PR[91] R[100]mm/sec CNT100;
   1:  CALL LASER_DRAHT_START;
   1:  PR[91,1] = PR[90,1] + -86.008;
   1:  PR[91,2] = PR[90,2] + -11.779;
   1:L PR[91] R[100]mm/sec CNT100;
   1:  PR[91,1] = PR[90,1] + -83.287;
   1:  PR[91,2] = PR[90,2] + -14.759;
   1:L PR[91] R[100]mm/sec CNT100;
   1:  PR[91,1] = PR[90,1] + -81.620;
   1:  PR[91,2] = PR[90,2] + -15.953;
   1:L PR[91] R[100]mm/sec CNT100;
   1:  PR[91,1] = PR[90,1] + -79.957;
   1:  PR[91,2] = PR[90,2] + -17.170;
   1:L PR[91] R[100]mm/sec CNT100;
   1:  PR[91,1] = PR[90,1] + -78.462;
   1:  PR[91,2] = PR[90,2] + -17.838;
   1:L PR[91] R[100]mm/sec CNT100;
   1:  PR[91,1] = PR[90,1] + -76.161;
   1:  PR[91,2] = PR[90,2] + -18.899;
   1:L PR[91] R[100]mm/sec CNT100;
   1:  PR[91,1] = PR[90,1] + -75.053;
   1:  PR[91,2] = PR[90,2] + -19.148;
   1:L PR[91] R[100]mm/sec CNT100;
   1:  PR[91,1] = PR[90,1] + -72.032;
   1:  PR[91,2] = PR[90,2] + -19.867;
   1:L PR[91] R[100]mm/sec CNT100;
   1:  PR[91,1] = PR[90,1] + -67.747;
   1:  PR[91,2] = PR[90,2] + -20.014;
   1:L PR[91] R[100]mm/sec CNT100;
   1:  PR[91,1] = PR[90,1] + -63.770;
   1:  PR[91,2] = PR[90,2] + -19.414;
   1:L PR[91] R[100]mm/sec CNT100;
   1:  PR[91,1] = PR[90,1] + -63.237;
   1:  PR[91,2] = PR[90,2] + -19.344;
   1:L PR[91] R[100]mm/sec CNT100;
   1:  PR[91,1] = PR[90,1] + -60.243;
   1:  PR[91,2] = PR[90,2] + -18.281;
   1:L PR[91] R[100]mm/sec CNT100;
   1:  PR[91,1] = PR[90,1] + -58.938;
   1:  PR[91,2] = PR[90,2] + -17.844;
   1:L PR[91] R[100]mm/sec CNT100;
   1:  PR[91,1] = PR[90,1] + -56.976;
   1:  PR[91,2] = PR[90,2] + -16.667;
   1:L PR[91] R[100]mm/sec CNT100;
   1:  PR[91,1] = PR[90,1] + -55.044;
   1:  PR[91,2] = PR[90,2] + -15.553;
   1:L PR[91] R[100]mm/sec CNT100;
   1:  PR[91,1] = PR[90,1] + -54.023;
   1:  PR[91,2] = PR[90,2] + -14.600;
   1:L PR[91] R[100]mm/sec CNT100;
   1:  PR[91,1] = PR[90,1] + -51.746;
   1:  PR[91,2] = PR[90,2] + -12.542;
   1:L PR[91] R[100]mm/sec CNT100;
   1:  PR[91,1] = PR[90,1] + -49.244;
   1:  PR[91,2] = PR[90,2] + -8.957;
   1:L PR[91] R[100]mm/sec CNT100;
   1:  PR[91,1] = PR[90,1] + -48.966;
   1:  PR[91,2] = PR[90,2] + -8.244;
   1:L PR[91] R[100]mm/sec CNT100;
   1:  PR[91,1] = PR[90,1] + -47.558;
   1:  PR[91,2] = PR[90,2] + -4.965;
   1:L PR[91] R[100]mm/sec CNT100;
   1:  PR[91,1] = PR[90,1] + -47.541;
   1:  PR[91,2] = PR[90,2] + -4.884;
   1:L PR[91] R[100]mm/sec CNT100;
   1:  PR[91,1] = PR[90,1] + -47.031;
   1:  PR[91,2] = PR[90,2] + -1.258;
   1:L PR[91] R[100]mm/sec CNT100;
   1:  PR[91,1] = PR[90,1] + -46.998;
   1:  PR[91,2] = PR[90,2] + -0.751;
   1:L PR[91] R[100]mm/sec CNT100;
   1:  PR[91,1] = PR[90,1] + -47.139;
   1:  PR[91,2] = PR[90,2] + 0.899;
   1:L PR[91] R[100]mm/sec CNT100;
   1:  PR[91,1] = PR[90,1] + -47.483;
   1:  PR[91,2] = PR[90,2] + 3.478;
   1:L PR[91] R[100]mm/sec CNT100;
   1:  PR[91,1] = PR[90,1] + -49.116;
   1:  PR[91,2] = PR[90,2] + 7.473;
   1:L PR[91] R[100]mm/sec CNT100;
   1:  PR[91,1] = PR[90,1] + -51.731;
   1:  PR[91,2] = PR[90,2] + 11.054;
   1:L PR[91] R[100]mm/sec CNT100;
   1:  PR[91,1] = PR[90,1] + -55.180;
   1:  PR[91,2] = PR[90,2] + 14.071;
   1:L PR[91] R[100]mm/sec CNT100;
   1:  PR[91,1] = PR[90,1] + -59.022;
   1:  PR[91,2] = PR[90,2] + 16.394;
   1:L PR[91] R[100]mm/sec CNT100;
   1:  PR[91,1] = PR[90,1] + -60.143;
   1:  PR[91,2] = PR[90,2] + 16.805;
   1:L PR[91] R[100]mm/sec CNT100;
   1:  PR[91,1] = PR[90,1] + -63.226;
   1:  PR[91,2] = PR[90,2] + 17.901;
   1:L PR[91] R[100]mm/sec CNT100;
   1:  PR[91,1] = PR[90,1] + -65.755;
   1:  PR[91,2] = PR[90,2] + 18.297;
   1:L PR[91] R[100]mm/sec CNT100;
   1:  PR[91,1] = PR[90,1] + -67.635;
   1:  PR[91,2] = PR[90,2] + 18.572;
   1:L PR[91] R[100]mm/sec CNT100;
   1:  PR[91,1] = PR[90,1] + -72.070;
   1:  PR[91,2] = PR[90,2] + 18.401;
   1:L PR[91] R[100]mm/sec CNT100;
   1:  PR[91,1] = PR[90,1] + -76.284;
   1:  PR[91,2] = PR[90,2] + 17.421;
   1:L PR[91] R[100]mm/sec CNT100;
   1:  PR[91,1] = PR[90,1] + -80.042;
   1:  PR[91,2] = PR[90,2] + 15.703;
   1:L PR[91] R[100]mm/sec CNT100;
   1:  PR[91,1] = PR[90,1] + -83.337;
   1:  PR[91,2] = PR[90,2] + 13.301;
   1:L PR[91] R[100]mm/sec CNT100;
   1:  PR[91,1] = PR[90,1] + -86.038;
   1:  PR[91,2] = PR[90,2] + 10.323;
   1:L PR[91] R[100]mm/sec CNT100;
   1:  PR[91,1] = PR[90,1] + -88.043;
   1:  PR[91,2] = PR[90,2] + 6.896;
   1:L PR[91] R[100]mm/sec CNT100;
   1:  PR[91,1] = PR[90,1] + -89.276;
   1:  PR[91,2] = PR[90,2] + 3.160;
   1:L PR[91] R[100]mm/sec CNT100;
   1:  PR[91,1] = PR[90,1] + -89.474;
   1:  PR[91,2] = PR[90,2] + 1.331;
   1:L PR[91] R[100]mm/sec CNT100;
   1:  PR[91,1] = PR[90,1] + -89.593;
   1:  PR[91,2] = PR[90,2] + 0.737;
   1:L PR[91] R[100]mm/sec CNT100;
   1:  PR[91,1] = PR[90,1] + -89.750;
   1:  PR[91,2] = PR[90,2] + -0.728;
   1:L PR[91] R[100]mm/sec CNT100;
   1:  PR[91,1] = PR[90,1] + -89.512;
   1:  PR[91,2] = PR[90,2] + -2.923;
   1:L PR[91] R[100]mm/sec CNT100;
   1:  PR[91,1] = PR[90,1] + -89.395;
   1:  PR[91,2] = PR[90,2] + -3.444;
   1:L PR[91] R[100]mm/sec CNT100;
   1:  PR[91,1] = PR[90,1] + -89.270;
   1:  PR[91,2] = PR[90,2] + -4.618;
   1:L PR[91] R[100]mm/sec CNT100;
   1:  PR[91,1] = PR[90,1] + -88.029;
   1:  PR[91,2] = PR[90,2] + -8.350;
   1:L PR[91] R[100]mm/sec CNT100TB   .50sec,CALL END_PUD;
   1:  PR[92] = PR[91];
   1:  PR[92,3] = PR[92,3] + 20;
   1:J PR[92] 10% FINE;
   1:  PR[91] = PR[90];
   1:  PR[91,1] = PR[90,1] + -0.522;
   1:  PR[91,2] = PR[90,2] + -2.915;
   1:  PR[91,3] = PR[90,3] + 37.895;
   1:  PR[92] = PR[91];
   1:  PR[92,3] = PR[92,3] + 20;
   1:J PR[92] 10% FINE;
   1:L PR[91] R[100]mm/sec CNT100;
   1:  CALL LASER_DRAHT_START;
   1:  PR[91,1] = PR[90,1] + -0.041;
   1:  PR[91,2] = PR[90,2] + -0.738;
   1:L PR[91] R[100]mm/sec CNT100;
   1:  PR[91,1] = PR[90,1] + -0.527;
   1:  PR[91,2] = PR[90,2] + 1.474;
   1:L PR[91] R[100]mm/sec CNT100;
   1:  PR[91,1] = PR[90,1] + -1.184;
   1:  PR[91,2] = PR[90,2] + 4.985;
   1:L PR[91] R[100]mm/sec CNT100;
   1:  PR[91,1] = PR[90,1] + -3.026;
   1:  PR[91,2] = PR[90,2] + 9.059;
   1:L PR[91] R[100]mm/sec CNT100;
   1:  PR[91,1] = PR[90,1] + -3.149;
   1:  PR[91,2] = PR[90,2] + 9.243;
   1:L PR[91] R[100]mm/sec CNT100;
   1:  PR[91,1] = PR[90,1] + -5.733;
   1:  PR[91,2] = PR[90,2] + 12.584;
   1:L PR[91] R[100]mm/sec CNT100;
   1:  PR[91,1] = PR[90,1] + -6.200;
   1:  PR[91,2] = PR[90,2] + 13.018;
   1:L PR[91] R[100]mm/sec CNT100;
   1:  PR[91,1] = PR[90,1] + -9.149;
   1:  PR[91,2] = PR[90,2] + 15.420;
   1:L PR[91] R[100]mm/sec CNT100;
   1:  PR[91,1] = PR[90,1] + -10.140;
   1:  PR[91,2] = PR[90,2] + 15.991;
   1:L PR[91] R[100]mm/sec CNT100;
   1:  PR[91,1] = PR[90,1] + -13.096;
   1:  PR[91,2] = PR[90,2] + 17.456;
   1:L PR[91] R[100]mm/sec CNT100;
   1:  PR[91,1] = PR[90,1] + -14.710;
   1:  PR[91,2] = PR[90,2] + 17.956;
   1:L PR[91] R[100]mm/sec CNT100;
   1:  PR[91,1] = PR[90,1] + -17.382;
   1:  PR[91,2] = PR[90,2] + 18.611;
   1:L PR[91] R[100]mm/sec CNT100;
   1:  PR[91,1] = PR[90,1] + -19.608;
   1:  PR[91,2] = PR[90,2] + 18.795;
   1:L PR[91] R[100]mm/sec CNT100;
   1:  PR[91,1] = PR[90,1] + -21.806;
   1:  PR[91,2] = PR[90,2] + 18.850;
   1:L PR[91] R[100]mm/sec CNT100;
   1:  PR[91,1] = PR[90,1] + -24.514;
   1:  PR[91,2] = PR[90,2] + 18.483;
   1:L PR[91] R[100]mm/sec CNT100;
   1:  PR[91,1] = PR[90,1] + -26.166;
   1:  PR[91,2] = PR[90,2] + 18.165;
   1:L PR[91] R[100]mm/sec CNT100;
   1:  PR[91,1] = PR[90,1] + -29.138;
   1:  PR[91,2] = PR[90,2] + 17.078;
   1:L PR[91] R[100]mm/sec CNT100;
   1:  PR[91,1] = PR[90,1] + -30.262;
   1:  PR[91,2] = PR[90,2] + 16.597;
   1:L PR[91] R[100]mm/sec CNT100;
   1:  PR[91,1] = PR[90,1] + -33.224;
   1:  PR[91,2] = PR[90,2] + 14.707;
   1:L PR[91] R[100]mm/sec CNT100;
   1:  PR[91,1] = PR[90,1] + -33.909;
   1:  PR[91,2] = PR[90,2] + 14.219;
   1:L PR[91] R[100]mm/sec CNT100;
   1:  PR[91,1] = PR[90,1] + -36.573;
   1:  PR[91,2] = PR[90,2] + 11.545;
   1:L PR[91] R[100]mm/sec CNT100;
   1:  PR[91,1] = PR[90,1] + -36.939;
   1:  PR[91,2] = PR[90,2] + 11.140;
   1:L PR[91] R[100]mm/sec CNT100;
   1:  PR[91,1] = PR[90,1] + -39.097;
   1:  PR[91,2] = PR[90,2] + 7.714;
   1:L PR[91] R[100]mm/sec CNT100;
   1:  PR[91,1] = PR[90,1] + -39.232;
   1:  PR[91,2] = PR[90,2] + 7.522;
   1:L PR[91] R[100]mm/sec CNT100;
   1:  PR[91,1] = PR[90,1] + -39.236;
   1:  PR[91,2] = PR[90,2] + 7.515;
   1:L PR[91] R[100]mm/sec CNT100;
   1:  PR[91,1] = PR[90,1] + -40.509;
   1:  PR[91,2] = PR[90,2] + 3.881;
   1:L PR[91] R[100]mm/sec CNT100;
   1:  PR[91,1] = PR[90,1] + -40.607;
   1:  PR[91,2] = PR[90,2] + 3.649;
   1:L PR[91] R[100]mm/sec CNT100;
   1:  PR[91,1] = PR[90,1] + -40.744;
   1:  PR[91,2] = PR[90,2] + 3.022;
   1:L PR[91] R[100]mm/sec CNT100;
   1:  PR[91,1] = PR[90,1] + -41.056;
   1:  PR[91,2] = PR[90,2] + 0.233;
   1:L PR[91] R[100]mm/sec CNT100;
   1:  PR[91,1] = PR[90,1] + -41.129;
   1:  PR[91,2] = PR[90,2] + -0.694;
   1:L PR[91] R[100]mm/sec CNT100;
   1:  PR[91,1] = PR[90,1] + -40.889;
   1:  PR[91,2] = PR[90,2] + -2.814;
   1:L PR[91] R[100]mm/sec CNT100;
   1:  PR[91,1] = PR[90,1] + -40.727;
   1:  PR[91,2] = PR[90,2] + -4.576;
   1:L PR[91] R[100]mm/sec CNT100;
   1:  PR[91,1] = PR[90,1] + -40.583;
   1:  PR[91,2] = PR[90,2] + -5.205;
   1:L PR[91] R[100]mm/sec CNT100;
   1:  PR[91,1] = PR[90,1] + -39.505;
   1:  PR[91,2] = PR[90,2] + -8.297;
   1:L PR[91] R[100]mm/sec CNT100;
   1:  PR[91,1] = PR[90,1] + -39.270;
   1:  PR[91,2] = PR[90,2] + -8.900;
   1:L PR[91] R[100]mm/sec CNT100;
   1:  PR[91,1] = PR[90,1] + -39.153;
   1:  PR[91,2] = PR[90,2] + -9.117;
   1:L PR[91] R[100]mm/sec CNT100;
   1:  PR[91,1] = PR[90,1] + -37.113;
   1:  PR[91,2] = PR[90,2] + -12.364;
   1:L PR[91] R[100]mm/sec CNT100;
   1:  PR[91,1] = PR[90,1] + -36.976;
   1:  PR[91,2] = PR[90,2] + -12.557;
   1:L PR[91] R[100]mm/sec CNT100;
   1:  PR[91,1] = PR[90,1] + -36.574;
   1:  PR[91,2] = PR[90,2] + -13.002;
   1:L PR[91] R[100]mm/sec CNT100;
   1:  PR[91,1] = PR[90,1] + -33.910;
   1:  PR[91,2] = PR[90,2] + -15.676;
   1:L PR[91] R[100]mm/sec CNT100;
   1:  PR[91,1] = PR[90,1] + -33.226;
   1:  PR[91,2] = PR[90,2] + -16.164;
   1:L PR[91] R[100]mm/sec CNT100;
   1:  PR[91,1] = PR[90,1] + -30.265;
   1:  PR[91,2] = PR[90,2] + -18.055;
   1:L PR[91] R[100]mm/sec CNT100;
   1:  PR[91,1] = PR[90,1] + -29.142;
   1:  PR[91,2] = PR[90,2] + -18.535;
   1:L PR[91] R[100]mm/sec CNT100;
   1:  PR[91,1] = PR[90,1] + -26.170;
   1:  PR[91,2] = PR[90,2] + -19.622;
   1:L PR[91] R[100]mm/sec CNT100;
   1:  PR[91,1] = PR[90,1] + -24.520;
   1:  PR[91,2] = PR[90,2] + -19.941;
   1:L PR[91] R[100]mm/sec CNT100;
   1:  PR[91,1] = PR[90,1] + -21.812;
   1:  PR[91,2] = PR[90,2] + -20.308;
   1:L PR[91] R[100]mm/sec CNT100;
   1:  PR[91,1] = PR[90,1] + -19.616;
   1:  PR[91,2] = PR[90,2] + -20.255;
   1:L PR[91] R[100]mm/sec CNT100;
   1:  PR[91,1] = PR[90,1] + -17.389;
   1:  PR[91,2] = PR[90,2] + -20.071;
   1:L PR[91] R[100]mm/sec CNT100;
   1:  PR[91,1] = PR[90,1] + -14.720;
   1:  PR[91,2] = PR[90,2] + -19.419;
   1:L PR[91] R[100]mm/sec CNT100;
   1:  PR[91,1] = PR[90,1] + -13.105;
   1:  PR[91,2] = PR[90,2] + -18.918;
   1:L PR[91] R[100]mm/sec CNT100;
   1:  PR[91,1] = PR[90,1] + -10.151;
   1:  PR[91,2] = PR[90,2] + -17.456;
   1:L PR[91] R[100]mm/sec CNT100;
   1:  PR[91,1] = PR[90,1] + -9.159;
   1:  PR[91,2] = PR[90,2] + -16.885;
   1:L PR[91] R[100]mm/sec CNT100;
   1:  PR[91,1] = PR[90,1] + -6.210;
   1:  PR[91,2] = PR[90,2] + -14.487;
   1:L PR[91] R[100]mm/sec CNT100;
   1:  PR[91,1] = PR[90,1] + -5.742;
   1:  PR[91,2] = PR[90,2] + -14.052;
   1:L PR[91] R[100]mm/sec CNT100;
   1:  PR[91,1] = PR[90,1] + -3.158;
   1:  PR[91,2] = PR[90,2] + -10.716;
   1:L PR[91] R[100]mm/sec CNT100;
   1:  PR[91,1] = PR[90,1] + -3.034;
   1:  PR[91,2] = PR[90,2] + -10.531;
   1:L PR[91] R[100]mm/sec CNT100;
   1:  PR[91,1] = PR[90,1] + -1.189;
   1:  PR[91,2] = PR[90,2] + -6.460;
   1:L PR[91] R[100]mm/sec CNT100;
   1:  PR[91,1] = PR[90,1] + -0.522;
   1:  PR[91,2] = PR[90,2] + -2.915;
   1:L PR[91] R[100]mm/sec CNT100TB   .50sec,CALL END_PUD;
   1:  PR[92] = PR[91];
   1:  PR[92,3] = PR[92,3] + 20;
   1:J PR[92] 10% FINE;
   1:  PR[91,1] = PR[90,1] + 3.385;
   1:  PR[91,2] = PR[90,2] + -0.662;
   1:  PR[92] = PR[91];
   1:  PR[92,3] = PR[92,3] + 20;
   1:J PR[92] 10% FINE;
   1:L PR[91] R[100]mm/sec CNT100;
   1:  CALL LASER_DRAHT_START;
   1:  PR[91,1] = PR[90,1] + 3.937;
   1:  PR[91,2] = PR[90,2] + -4.586;
   1:L PR[91] R[100]mm/sec CNT100;
   1:  PR[91,1] = PR[90,1] + 4.284;
   1:  PR[91,2] = PR[90,2] + -6.155;
   1:L PR[91] R[100]mm/sec CNT100;
   1:  PR[91,1] = PR[90,1] + 5.697;
   1:  PR[91,2] = PR[90,2] + -9.537;
   1:L PR[91] R[100]mm/sec CNT100;
   1:  PR[91,1] = PR[90,1] + 6.139;
   1:  PR[91,2] = PR[90,2] + -10.641;
   1:L PR[91] R[100]mm/sec CNT100;
   1:  PR[91,1] = PR[90,1] + 6.266;
   1:  PR[91,2] = PR[90,2] + -10.893;
   1:L PR[91] R[100]mm/sec CNT100;
   1:  PR[91,1] = PR[90,1] + 9.333;
   1:  PR[91,2] = PR[90,2] + -14.856;
   1:L PR[91] R[100]mm/sec CNT100;
   1:  PR[91,1] = PR[90,1] + 9.433;
   1:  PR[91,2] = PR[90,2] + -14.999;
   1:L PR[91] R[100]mm/sec CNT100;
   1:  PR[91,1] = PR[90,1] + 9.569;
   1:  PR[91,2] = PR[90,2] + -15.142;
   1:L PR[91] R[100]mm/sec CNT100;
   1:  PR[91,1] = PR[90,1] + 13.652;
   1:  PR[91,2] = PR[90,2] + -18.238;
   1:L PR[91] R[100]mm/sec CNT100;
   1:  PR[91,1] = PR[90,1] + 13.755;
   1:  PR[91,2] = PR[90,2] + -18.302;
   1:L PR[91] R[100]mm/sec CNT100;
   1:  PR[91,1] = PR[90,1] + 18.614;
   1:  PR[91,2] = PR[90,2] + -20.286;
   1:L PR[91] R[100]mm/sec CNT100;
   1:  PR[91,1] = PR[90,1] + 23.877;
   1:  PR[91,2] = PR[90,2] + -20.954;
   1:L PR[91] R[100]mm/sec CNT100;
   1:  PR[91,1] = PR[90,1] + 29.070;
   1:  PR[91,2] = PR[90,2] + -20.267;
   1:L PR[91] R[100]mm/sec CNT100;
   1:  PR[91,1] = PR[90,1] + 33.921;
   1:  PR[91,2] = PR[90,2] + -18.278;
   1:L PR[91] R[100]mm/sec CNT100;
   1:  PR[91,1] = PR[90,1] + 38.090;
   1:  PR[91,2] = PR[90,2] + -15.120;
   1:L PR[91] R[100]mm/sec CNT100;
   1:  PR[91,1] = PR[90,1] + 41.369;
   1:  PR[91,2] = PR[90,2] + -10.919;
   1:L PR[91] R[100]mm/sec CNT100;
   1:  PR[91,1] = PR[90,1] + 42.983;
   1:  PR[91,2] = PR[90,2] + -7.976;
   1:L PR[91] R[100]mm/sec CNT100;
   1:  PR[91,1] = PR[90,1] + 45.288;
   1:  PR[91,2] = PR[90,2] + -10.358;
   1:L PR[91] R[100]mm/sec CNT100;
   1:  PR[91,1] = PR[90,1] + 47.970;
   1:  PR[91,2] = PR[90,2] + -13.572;
   1:L PR[91] R[100]mm/sec CNT100;
   1:  PR[91,1] = PR[90,1] + 48.885;
   1:  PR[91,2] = PR[90,2] + -14.529;
   1:L PR[91] R[100]mm/sec CNT100;
   1:  PR[91,1] = PR[90,1] + 51.335;
   1:  PR[91,2] = PR[90,2] + -16.321;
   1:L PR[91] R[100]mm/sec CNT100;
   1:  PR[91,1] = PR[90,1] + 54.397;
   1:  PR[91,2] = PR[90,2] + -18.210;
   1:L PR[91] R[100]mm/sec CNT100;
   1:  PR[91,1] = PR[90,1] + 55.333;
   1:  PR[91,2] = PR[90,2] + -18.619;
   1:L PR[91] R[100]mm/sec CNT100;
   1:  PR[91,1] = PR[90,1] + 57.990;
   1:  PR[91,2] = PR[90,2] + -19.512;
   1:L PR[91] R[100]mm/sec CNT100;
   1:  PR[91,1] = PR[90,1] + 60.242;
   1:  PR[91,2] = PR[90,2] + -20.391;
   1:L PR[91] R[100]mm/sec CNT100;
   1:  PR[91,1] = PR[90,1] + 60.870;
   1:  PR[91,2] = PR[90,2] + -20.545;
   1:L PR[91] R[100]mm/sec CNT100;
   1:  PR[91,1] = PR[90,1] + 65.019;
   1:  PR[91,2] = PR[90,2] + -21.162;
   1:L PR[91] R[100]mm/sec CNT100;
   1:  PR[91,1] = PR[90,1] + 67.358;
   1:  PR[91,2] = PR[90,2] + -21.246;
   1:L PR[91] R[100]mm/sec CNT100;
   1:  PR[91,1] = PR[90,1] + 69.662;
   1:  PR[91,2] = PR[90,2] + -21.085;
   1:L PR[91] R[100]mm/sec CNT100;
   1:  PR[91,1] = PR[90,1] + 73.257;
   1:  PR[91,2] = PR[90,2] + -20.487;
   1:L PR[91] R[100]mm/sec CNT100;
   1:  PR[91,1] = PR[90,1] + 74.066;
   1:  PR[91,2] = PR[90,2] + -20.249;
   1:L PR[91] R[100]mm/sec CNT100;
   1:  PR[91,1] = PR[90,1] + 78.258;
   1:  PR[91,2] = PR[90,2] + -18.646;
   1:L PR[91] R[100]mm/sec CNT100;
   1:  PR[91,1] = PR[90,1] + 82.107;
   1:  PR[91,2] = PR[90,2] + -16.130;
   1:L PR[91] R[100]mm/sec CNT100;
   1:  PR[91,1] = PR[90,1] + 85.274;
   1:  PR[91,2] = PR[90,2] + -12.918;
   1:L PR[91] R[100]mm/sec CNT100;
   1:  PR[91,1] = PR[90,1] + 87.630;
   1:  PR[91,2] = PR[90,2] + -9.162;
   1:L PR[91] R[100]mm/sec CNT100;
   1:  PR[91,1] = PR[90,1] + 88.097;
   1:  PR[91,2] = PR[90,2] + -7.845;
   1:L PR[91] R[100]mm/sec CNT100;
   1:  PR[91,1] = PR[90,1] + 89.077;
   1:  PR[91,2] = PR[90,2] + -5.041;
   1:L PR[91] R[100]mm/sec CNT100;
   1:  PR[91,1] = PR[90,1] + 89.568;
   1:  PR[91,2] = PR[90,2] + -0.729;
   1:L PR[91] R[100]mm/sec CNT100;
   1:  PR[91,1] = PR[90,1] + 89.077;
   1:  PR[91,2] = PR[90,2] + 3.581;
   1:L PR[91] R[100]mm/sec CNT100;
   1:  PR[91,1] = PR[90,1] + 87.628;
   1:  PR[91,2] = PR[90,2] + 7.706;
   1:L PR[91] R[100]mm/sec CNT100;
   1:  PR[91,1] = PR[90,1] + 85.279;
   1:  PR[91,2] = PR[90,2] + 11.451;
   1:L PR[91] R[100]mm/sec CNT100;
   1:  PR[91,1] = PR[90,1] + 84.620;
   1:  PR[91,2] = PR[90,2] + 12.107;
   1:L PR[91] R[100]mm/sec CNT100;
   1:  PR[91,1] = PR[90,1] + 82.105;
   1:  PR[91,2] = PR[90,2] + 14.672;
   1:L PR[91] R[100]mm/sec CNT100;
   1:  PR[91,1] = PR[90,1] + 78.258;
   1:  PR[91,2] = PR[90,2] + 17.187;
   1:L PR[91] R[100]mm/sec CNT100;
   1:  PR[91,1] = PR[90,1] + 74.066;
   1:  PR[91,2] = PR[90,2] + 18.790;
   1:L PR[91] R[100]mm/sec CNT100;
   1:  PR[91,1] = PR[90,1] + 73.257;
   1:  PR[91,2] = PR[90,2] + 19.028;
   1:L PR[91] R[100]mm/sec CNT100;
   1:  PR[91,1] = PR[90,1] + 69.663;
   1:  PR[91,2] = PR[90,2] + 19.626;
   1:L PR[91] R[100]mm/sec CNT100;
   1:  PR[91,1] = PR[90,1] + 67.359;
   1:  PR[91,2] = PR[90,2] + 19.787;
   1:L PR[91] R[100]mm/sec CNT100;
   1:  PR[91,1] = PR[90,1] + 65.019;
   1:  PR[91,2] = PR[90,2] + 19.703;
   1:L PR[91] R[100]mm/sec CNT100;
   1:  PR[91,1] = PR[90,1] + 60.872;
   1:  PR[91,2] = PR[90,2] + 19.086;
   1:L PR[91] R[100]mm/sec CNT100;
   1:  PR[91,1] = PR[90,1] + 60.243;
   1:  PR[91,2] = PR[90,2] + 18.933;
   1:L PR[91] R[100]mm/sec CNT100;
   1:  PR[91,1] = PR[90,1] + 57.989;
   1:  PR[91,2] = PR[90,2] + 18.053;
   1:L PR[91] R[100]mm/sec CNT100;
   1:  PR[91,1] = PR[90,1] + 55.325;
   1:  PR[91,2] = PR[90,2] + 17.158;
   1:L PR[91] R[100]mm/sec CNT100;
   1:  PR[91,1] = PR[90,1] + 54.374;
   1:  PR[91,2] = PR[90,2] + 16.739;
   1:L PR[91] R[100]mm/sec CNT100;
   1:  PR[91,1] = PR[90,1] + 51.306;
   1:  PR[91,2] = PR[90,2] + 14.848;
   1:L PR[91] R[100]mm/sec CNT100;
   1:  PR[91,1] = PR[90,1] + 48.827;
   1:  PR[91,2] = PR[90,2] + 13.016;
   1:L PR[91] R[100]mm/sec CNT100;
   1:  PR[91,1] = PR[90,1] + 47.925;
   1:  PR[91,2] = PR[90,2] + 12.075;
   1:L PR[91] R[100]mm/sec CNT100;
   1:  PR[91,1] = PR[90,1] + 45.441;
   1:  PR[91,2] = PR[90,2] + 9.058;
   1:L PR[91] R[100]mm/sec CNT100;
   1:  PR[91,1] = PR[90,1] + 42.979;
   1:  PR[91,2] = PR[90,2] + 6.500;
   1:L PR[91] R[100]mm/sec CNT100;
   1:  PR[91,1] = PR[90,1] + 41.357;
   1:  PR[91,2] = PR[90,2] + 9.483;
   1:L PR[91] R[100]mm/sec CNT100;
   1:  PR[91,1] = PR[90,1] + 41.222;
   1:  PR[91,2] = PR[90,2] + 9.669;
   1:L PR[91] R[100]mm/sec CNT100;
   1:  PR[91,1] = PR[90,1] + 38.058;
   1:  PR[91,2] = PR[90,2] + 13.693;
   1:L PR[91] R[100]mm/sec CNT100;
   1:  PR[91,1] = PR[90,1] + 33.885;
   1:  PR[91,2] = PR[90,2] + 16.840;
   1:L PR[91] R[100]mm/sec CNT100;
   1:  PR[91,1] = PR[90,1] + 29.034;
   1:  PR[91,2] = PR[90,2] + 18.817;
   1:L PR[91] R[100]mm/sec CNT100;
   1:  PR[91,1] = PR[90,1] + 23.845;
   1:  PR[91,2] = PR[90,2] + 19.495;
   1:L PR[91] R[100]mm/sec CNT100;
   1:  PR[91,1] = PR[90,1] + 18.587;
   1:  PR[91,2] = PR[90,2] + 18.820;
   1:L PR[91] R[100]mm/sec CNT100;
   1:  PR[91,1] = PR[90,1] + 13.737;
   1:  PR[91,2] = PR[90,2] + 16.833;
   1:L PR[91] R[100]mm/sec CNT100;
   1:  PR[91,1] = PR[90,1] + 13.634;
   1:  PR[91,2] = PR[90,2] + 16.769;
   1:L PR[91] R[100]mm/sec CNT100;
   1:  PR[91,1] = PR[90,1] + 9.558;
   1:  PR[91,2] = PR[90,2] + 13.673;
   1:L PR[91] R[100]mm/sec CNT100;
   1:  PR[91,1] = PR[90,1] + 9.386;
   1:  PR[91,2] = PR[90,2] + 13.492;
   1:L PR[91] R[100]mm/sec CNT100;
   1:  PR[91,1] = PR[90,1] + 6.330;
   1:  PR[91,2] = PR[90,2] + 9.542;
   1:L PR[91] R[100]mm/sec CNT100;
   1:  PR[91,1] = PR[90,1] + 6.175;
   1:  PR[91,2] = PR[90,2] + 9.261;
   1:L PR[91] R[100]mm/sec CNT100;
   1:  PR[91,1] = PR[90,1] + 4.295;
   1:  PR[91,2] = PR[90,2] + 4.736;
   1:L PR[91] R[100]mm/sec CNT100;
   1:  PR[91,1] = PR[90,1] + 3.947;
   1:  PR[91,2] = PR[90,2] + 3.180;
   1:L PR[91] R[100]mm/sec CNT100;
   1:  PR[91,1] = PR[90,1] + 3.727;
   1:  PR[91,2] = PR[90,2] + 1.543;
   1:L PR[91] R[100]mm/sec CNT100;
   1:  PR[91,1] = PR[90,1] + 3.385;
   1:  PR[91,2] = PR[90,2] + -0.662;
   1:L PR[91] R[100]mm/sec CNT100TB   .50sec,CALL END_PUD;
   1:  PR[92] = PR[91];
   1:  PR[92,3] = PR[92,3] + 20;
   1:J PR[92] 10% FINE;
   1:  PR[91,1] = PR[90,1] + -48.280;
   1:  PR[91,2] = PR[90,2] + -9.189;
   1:  PR[92] = PR[91];
   1:  PR[92,3] = PR[92,3] + 20;
   1:J PR[92] 10% FINE;
   1:L PR[91] R[100]mm/sec CNT100;
   1:  CALL LASER_DRAHT_START;
   1:  PR[91,1] = PR[90,1] + -47.842;
   1:  PR[91,2] = PR[90,2] + -8.344;
   1:L PR[91] R[100]mm/sec CNT100;
   1:  PR[91,1] = PR[90,1] + -46.537;
   1:  PR[91,2] = PR[90,2] + -5.304;
   1:L PR[91] R[100]mm/sec CNT100;
   1:  PR[91,1] = PR[90,1] + -46.350;
   1:  PR[91,2] = PR[90,2] + -4.422;
   1:L PR[91] R[100]mm/sec CNT100;
   1:  PR[91,1] = PR[90,1] + -46.052;
   1:  PR[91,2] = PR[90,2] + -2.307;
   1:L PR[91] R[100]mm/sec CNT100;
   1:  PR[91,1] = PR[90,1] + -45.952;
   1:  PR[91,2] = PR[90,2] + -0.751;
   1:L PR[91] R[100]mm/sec CNT100;
   1:  PR[91,1] = PR[90,1] + -45.988;
   1:  PR[91,2] = PR[90,2] + -0.330;
   1:L PR[91] R[100]mm/sec CNT100;
   1:  PR[91,1] = PR[90,1] + -46.502;
   1:  PR[91,2] = PR[90,2] + 3.527;
   1:L PR[91] R[100]mm/sec CNT100;
   1:  PR[91,1] = PR[90,1] + -48.161;
   1:  PR[91,2] = PR[90,2] + 7.565;
   1:L PR[91] R[100]mm/sec CNT100;
   1:  PR[91,1] = PR[90,1] + -50.814;
   1:  PR[91,2] = PR[90,2] + 11.180;
   1:L PR[91] R[100]mm/sec CNT100;
   1:  PR[91,1] = PR[90,1] + -54.291;
   1:  PR[91,2] = PR[90,2] + 14.198;
   1:L PR[91] R[100]mm/sec CNT100;
   1:  PR[91,1] = PR[90,1] + -57.643;
   1:  PR[91,2] = PR[90,2] + 16.065;
   1:L PR[91] R[100]mm/sec CNT100;
   1:  PR[91,1] = PR[90,1] + -58.400;
   1:  PR[91,2] = PR[90,2] + 16.522;
   1:L PR[91] R[100]mm/sec CNT100;
   1:  PR[91,1] = PR[90,1] + -62.648;
   1:  PR[91,2] = PR[90,2] + 18.035;
   1:L PR[91] R[100]mm/sec CNT100;
   1:  PR[91,1] = PR[90,1] + -64.155;
   1:  PR[91,2] = PR[90,2] + 18.271;
   1:L PR[91] R[100]mm/sec CNT100;
   1:  PR[91,1] = PR[90,1] + -67.091;
   1:  PR[91,2] = PR[90,2] + 18.701;
   1:L PR[91] R[100]mm/sec CNT100;
   1:  PR[91,1] = PR[90,1] + -69.914;
   1:  PR[91,2] = PR[90,2] + 18.597;
   1:L PR[91] R[100]mm/sec CNT100;
   1:  PR[91,1] = PR[90,1] + -71.543;
   1:  PR[91,2] = PR[90,2] + 18.521;
   1:L PR[91] R[100]mm/sec CNT100;
   1:  PR[91,1] = PR[90,1] + -75.829;
   1:  PR[91,2] = PR[90,2] + 17.518;
   1:L PR[91] R[100]mm/sec CNT100;
   1:  PR[91,1] = PR[90,1] + -79.715;
   1:  PR[91,2] = PR[90,2] + 15.766;
   1:L PR[91] R[100]mm/sec CNT100;
   1:  PR[91,1] = PR[90,1] + -83.016;
   1:  PR[91,2] = PR[90,2] + 13.356;
   1:L PR[91] R[100]mm/sec CNT100;
   1:  PR[91,1] = PR[90,1] + -85.724;
   1:  PR[91,2] = PR[90,2] + 10.364;
   1:L PR[91] R[100]mm/sec CNT100;
   1:  PR[91,1] = PR[90,1] + -87.735;
   1:  PR[91,2] = PR[90,2] + 6.923;
   1:L PR[91] R[100]mm/sec CNT100;
   1:  PR[91,1] = PR[90,1] + -88.971;
   1:  PR[91,2] = PR[90,2] + 3.173;
   1:L PR[91] R[100]mm/sec CNT100;
   1:  PR[91,1] = PR[90,1] + -89.113;
   1:  PR[91,2] = PR[90,2] + 1.861;
   1:L PR[91] R[100]mm/sec CNT100;
   1:  PR[91,1] = PR[90,1] + -89.201;
   1:  PR[91,2] = PR[90,2] + 1.425;
   1:L PR[91] R[100]mm/sec CNT100;
   1:  PR[91,1] = PR[90,1] + -89.431;
   1:  PR[91,2] = PR[90,2] + -0.728;
   1:L PR[91] R[100]mm/sec CNT100;
   1:  PR[91,1] = PR[90,1] + -89.263;
   1:  PR[91,2] = PR[90,2] + -2.277;
   1:L PR[91] R[100]mm/sec CNT100;
   1:  PR[91,1] = PR[90,1] + -89.103;
   1:  PR[91,2] = PR[90,2] + -2.989;
   1:L PR[91] R[100]mm/sec CNT100;
   1:  PR[91,1] = PR[90,1] + -88.928;
   1:  PR[91,2] = PR[90,2] + -4.633;
   1:L PR[91] R[100]mm/sec CNT100;
   1:  PR[91,1] = PR[90,1] + -87.684;
   1:  PR[91,2] = PR[90,2] + -8.380;
   1:L PR[91] R[100]mm/sec CNT100;
   1:  PR[91,1] = PR[90,1] + -85.656;
   1:  PR[91,2] = PR[90,2] + -11.824;
   1:L PR[91] R[100]mm/sec CNT100;
   1:  PR[91,1] = PR[90,1] + -82.928;
   1:  PR[91,2] = PR[90,2] + -14.818;
   1:L PR[91] R[100]mm/sec CNT100;
   1:  PR[91,1] = PR[90,1] + -81.651;
   1:  PR[91,2] = PR[90,2] + -15.733;
   1:L PR[91] R[100]mm/sec CNT100;
   1:  PR[91,1] = PR[90,1] + -79.588;
   1:  PR[91,2] = PR[90,2] + -17.243;
   1:L PR[91] R[100]mm/sec CNT100;
   1:  PR[91,1] = PR[90,1] + -78.546;
   1:  PR[91,2] = PR[90,2] + -17.708;
   1:L PR[91] R[100]mm/sec CNT100;
   1:  PR[91,1] = PR[90,1] + -75.767;
   1:  PR[91,2] = PR[90,2] + -18.989;
   1:L PR[91] R[100]mm/sec CNT100;
   1:  PR[91,1] = PR[90,1] + -71.625;
   1:  PR[91,2] = PR[90,2] + -19.966;
   1:L PR[91] R[100]mm/sec CNT100;
   1:  PR[91,1] = PR[90,1] + -67.146;
   1:  PR[91,2] = PR[90,2] + -20.149;
   1:L PR[91] R[100]mm/sec CNT100;
   1:  PR[91,1] = PR[90,1] + -63.769;
   1:  PR[91,2] = PR[90,2] + -19.645;
   1:L PR[91] R[100]mm/sec CNT100;
   1:  PR[91,1] = PR[90,1] + -62.587;
   1:  PR[91,2] = PR[90,2] + -19.490;
   1:L PR[91] R[100]mm/sec CNT100;
   1:  PR[91,1] = PR[90,1] + -60.217;
   1:  PR[91,2] = PR[90,2] + -18.649;
   1:L PR[91] R[100]mm/sec CNT100;
   1:  PR[91,1] = PR[90,1] + -58.248;
   1:  PR[91,2] = PR[90,2] + -17.990;
   1:L PR[91] R[100]mm/sec CNT100;
   1:  PR[91,1] = PR[90,1] + -56.891;
   1:  PR[91,2] = PR[90,2] + -17.175;
   1:L PR[91] R[100]mm/sec CNT100;
   1:  PR[91,1] = PR[90,1] + -54.312;
   1:  PR[91,2] = PR[90,2] + -15.689;
   1:L PR[91] R[100]mm/sec CNT100;
   1:  PR[91,1] = PR[90,1] + -53.842;
   1:  PR[91,2] = PR[90,2] + -15.250;
   1:L PR[91] R[100]mm/sec CNT100;
   1:  PR[91,1] = PR[90,1] + -50.938;
   1:  PR[91,2] = PR[90,2] + -12.631;
   1:L PR[91] R[100]mm/sec CNT100;
   1:  PR[91,1] = PR[90,1] + -48.280;
   1:  PR[91,2] = PR[90,2] + -9.189;
   1:L PR[91] R[100]mm/sec CNT100TB   .50sec,CALL END_PUD;
   1:  PR[92] = PR[91];
   1:  PR[92,3] = PR[92,3] + 20;
   1:J PR[92] 10% FINE;
   1:  PR[91] = PR[90];
   1:  PR[91,1] = PR[90,1] + -47.207;
   1:  PR[91,2] = PR[90,2] + 7.658;
   1:  PR[91,3] = PR[90,3] + 39.195;
   1:  PR[92] = PR[91];
   1:  PR[92,3] = PR[92,3] + 20;
   1:J PR[92] 10% FINE;
   1:L PR[91] R[100]mm/sec CNT100;
   1:  CALL LASER_DRAHT_START;
   1:  PR[91,1] = PR[90,1] + -49.902;
   1:  PR[91,2] = PR[90,2] + 11.311;
   1:L PR[91] R[100]mm/sec CNT100;
   1:  PR[91,1] = PR[90,1] + -51.244;
   1:  PR[91,2] = PR[90,2] + 12.483;
   1:L PR[91] R[100]mm/sec CNT100;
   1:  PR[91,1] = PR[90,1] + -53.419;
   1:  PR[91,2] = PR[90,2] + 14.347;
   1:L PR[91] R[100]mm/sec CNT100;
   1:  PR[91,1] = PR[90,1] + -57.577;
   1:  PR[91,2] = PR[90,2] + 16.651;
   1:L PR[91] R[100]mm/sec CNT100;
   1:  PR[91,1] = PR[90,1] + -60.018;
   1:  PR[91,2] = PR[90,2] + 17.440;
   1:L PR[91] R[100]mm/sec CNT100;
   1:  PR[91,1] = PR[90,1] + -62.061;
   1:  PR[91,2] = PR[90,2] + 18.166;
   1:L PR[91] R[100]mm/sec CNT100;
   1:  PR[91,1] = PR[90,1] + -66.547;
   1:  PR[91,2] = PR[90,2] + 18.829;
   1:L PR[91] R[100]mm/sec CNT100;
   1:  PR[91,1] = PR[90,1] + -68.412;
   1:  PR[91,2] = PR[90,2] + 18.760;
   1:L PR[91] R[100]mm/sec CNT100;
   1:  PR[91,1] = PR[90,1] + -71.023;
   1:  PR[91,2] = PR[90,2] + 18.639;
   1:L PR[91] R[100]mm/sec CNT100;
   1:  PR[91,1] = PR[90,1] + -75.333;
   1:  PR[91,2] = PR[90,2] + 17.623;
   1:L PR[91] R[100]mm/sec CNT100;
   1:  PR[91,1] = PR[90,1] + -79.285;
   1:  PR[91,2] = PR[90,2] + 15.844;
   1:L PR[91] R[100]mm/sec CNT100;
   1:  PR[91,1] = PR[90,1] + -82.702;
   1:  PR[91,2] = PR[90,2] + 13.402;
   1:L PR[91] R[100]mm/sec CNT100;
   1:  PR[91,1] = PR[90,1] + -85.411;
   1:  PR[91,2] = PR[90,2] + 10.405;
   1:L PR[91] R[100]mm/sec CNT100;
   1:  PR[91,1] = PR[90,1] + -87.427;
   1:  PR[91,2] = PR[90,2] + 6.951;
   1:L PR[91] R[100]mm/sec CNT100;
   1:  PR[91,1] = PR[90,1] + -88.666;
   1:  PR[91,2] = PR[90,2] + 3.187;
   1:L PR[91] R[100]mm/sec CNT100;
   1:  PR[91,1] = PR[90,1] + -88.752;
   1:  PR[91,2] = PR[90,2] + 2.391;
   1:L PR[91] R[100]mm/sec CNT100;
   1:  PR[91,1] = PR[90,1] + -88.808;
   1:  PR[91,2] = PR[90,2] + 2.113;
   1:L PR[91] R[100]mm/sec CNT100;
   1:  PR[91,1] = PR[90,1] + -89.112;
   1:  PR[91,2] = PR[90,2] + -0.728;
   1:L PR[91] R[100]mm/sec CNT100;
   1:  PR[91,1] = PR[90,1] + -89.014;
   1:  PR[91,2] = PR[90,2] + -1.630;
   1:L PR[91] R[100]mm/sec CNT100;
   1:  PR[91,1] = PR[90,1] + -88.812;
   1:  PR[91,2] = PR[90,2] + -2.533;
   1:L PR[91] R[100]mm/sec CNT100;
   1:  PR[91,1] = PR[90,1] + -88.586;
   1:  PR[91,2] = PR[90,2] + -4.648;
   1:L PR[91] R[100]mm/sec CNT100;
   1:  PR[91,1] = PR[90,1] + -87.339;
   1:  PR[91,2] = PR[90,2] + -8.411;
   1:L PR[91] R[100]mm/sec CNT100;
   1:  PR[91,1] = PR[90,1] + -85.305;
   1:  PR[91,2] = PR[90,2] + -11.869;
   1:L PR[91] R[100]mm/sec CNT100;
   1:  PR[91,1] = PR[90,1] + -82.564;
   1:  PR[91,2] = PR[90,2] + -14.882;
   1:L PR[91] R[100]mm/sec CNT100;
   1:  PR[91,1] = PR[90,1] + -79.213;
   1:  PR[91,2] = PR[90,2] + -17.320;
   1:L PR[91] R[100]mm/sec CNT100;
   1:  PR[91,1] = PR[90,1] + -75.385;
   1:  PR[91,2] = PR[90,2] + -19.075;
   1:L PR[91] R[100]mm/sec CNT100;
   1:  PR[91,1] = PR[90,1] + -71.106;
   1:  PR[91,2] = PR[90,2] + -20.083;
   1:L PR[91] R[100]mm/sec CNT100;
   1:  PR[91,1] = PR[90,1] + -67.492;
   1:  PR[91,2] = PR[90,2] + -20.230;
   1:L PR[91] R[100]mm/sec CNT100;
   1:  PR[91,1] = PR[90,1] + -66.515;
   1:  PR[91,2] = PR[90,2] + -20.286;
   1:L PR[91] R[100]mm/sec CNT100;
   1:  PR[91,1] = PR[90,1] + -63.770;
   1:  PR[91,2] = PR[90,2] + -19.876;
   1:L PR[91] R[100]mm/sec CNT100;
   1:  PR[91,1] = PR[90,1] + -61.937;
   1:  PR[91,2] = PR[90,2] + -19.636;
   1:L PR[91] R[100]mm/sec CNT100;
   1:  PR[91,1] = PR[90,1] + -60.190;
   1:  PR[91,2] = PR[90,2] + -19.016;
   1:L PR[91] R[100]mm/sec CNT100;
   1:  PR[91,1] = PR[90,1] + -57.558;
   1:  PR[91,2] = PR[90,2] + -18.135;
   1:L PR[91] R[100]mm/sec CNT100;
   1:  PR[91,1] = PR[90,1] + -56.806;
   1:  PR[91,2] = PR[90,2] + -17.684;
   1:L PR[91] R[100]mm/sec CNT100;
   1:  PR[91,1] = PR[90,1] + -53.568;
   1:  PR[91,2] = PR[90,2] + -15.818;
   1:L PR[91] R[100]mm/sec CNT100;
   1:  PR[91,1] = PR[90,1] + -53.267;
   1:  PR[91,2] = PR[90,2] + -15.544;
   1:L PR[91] R[100]mm/sec CNT100;
   1:  PR[91,1] = PR[90,1] + -50.100;
   1:  PR[91,2] = PR[90,2] + -12.951;
   1:L PR[91] R[100]mm/sec CNT100;
   1:  PR[91,1] = PR[90,1] + -49.327;
   1:  PR[91,2] = PR[90,2] + -12.096;
   1:L PR[91] R[100]mm/sec CNT100;
   1:  PR[91,1] = PR[90,1] + -47.391;
   1:  PR[91,2] = PR[90,2] + -9.587;
   1:L PR[91] R[100]mm/sec CNT100;
   1:  PR[91,1] = PR[90,1] + -46.330;
   1:  PR[91,2] = PR[90,2] + -7.540;
   1:L PR[91] R[100]mm/sec CNT100;
   1:  PR[91,1] = PR[90,1] + -45.515;
   1:  PR[91,2] = PR[90,2] + -5.643;
   1:L PR[91] R[100]mm/sec CNT100;
   1:  PR[91,1] = PR[90,1] + -45.158;
   1:  PR[91,2] = PR[90,2] + -3.960;
   1:L PR[91] R[100]mm/sec CNT100;
   1:  PR[91,1] = PR[90,1] + -45.073;
   1:  PR[91,2] = PR[90,2] + -3.355;
   1:L PR[91] R[100]mm/sec CNT100;
   1:  PR[91,1] = PR[90,1] + -45.003;
   1:  PR[91,2] = PR[90,2] + -2.254;
   1:L PR[91] R[100]mm/sec CNT100;
   1:  PR[91,1] = PR[90,1] + -44.855;
   1:  PR[91,2] = PR[90,2] + -0.642;
   1:L PR[91] R[100]mm/sec CNT100;
   1:  PR[91,1] = PR[90,1] + -45.345;
   1:  PR[91,2] = PR[90,2] + 3.088;
   1:L PR[91] R[100]mm/sec CNT100;
   1:  PR[91,1] = PR[90,1] + -45.463;
   1:  PR[91,2] = PR[90,2] + 3.590;
   1:L PR[91] R[100]mm/sec CNT100;
   1:  PR[91,1] = PR[90,1] + -46.247;
   1:  PR[91,2] = PR[90,2] + 5.331;
   1:L PR[91] R[100]mm/sec CNT100;
   1:  PR[91,1] = PR[90,1] + -47.206;
   1:  PR[91,2] = PR[90,2] + 7.658;
   1:L PR[91] R[100]mm/sec CNT100TB   .50sec,CALL END_PUD;
   1:  PR[92] = PR[91];
   1:  PR[92,3] = PR[92,3] + 20;
   1:J PR[92] 10% FINE;
   1:  PR[91,1] = PR[90,1] + -40.199;
   1:  PR[91,2] = PR[90,2] + 4.341;
   1:  PR[92] = PR[91];
   1:  PR[92,3] = PR[92,3] + 20;
   1:J PR[92] 10% FINE;
   1:L PR[91] R[100]mm/sec CNT100;
   1:  CALL LASER_DRAHT_START;
   1:  PR[91,1] = PR[90,1] + -40.331;
   1:  PR[91,2] = PR[90,2] + 4.012;
   1:L PR[91] R[100]mm/sec CNT100;
   1:  PR[91,1] = PR[90,1] + -40.685;
   1:  PR[91,2] = PR[90,2] + 2.385;
   1:L PR[91] R[100]mm/sec CNT100;
   1:  PR[91,1] = PR[90,1] + -40.769;
   1:  PR[91,2] = PR[90,2] + 1.636;
   1:L PR[91] R[100]mm/sec CNT100;
   1:  PR[91,1] = PR[90,1] + -40.955;
   1:  PR[91,2] = PR[90,2] + -0.751;
   1:L PR[91] R[100]mm/sec CNT100;
   1:  PR[91,1] = PR[90,1] + -40.654;
   1:  PR[91,2] = PR[90,2] + -4.032;
   1:L PR[91] R[100]mm/sec CNT100;
   1:  PR[91,1] = PR[90,1] + -40.296;
   1:  PR[91,2] = PR[90,2] + -5.597;
   1:L PR[91] R[100]mm/sec CNT100;
   1:  PR[91,1] = PR[90,1] + -39.609;
   1:  PR[91,2] = PR[90,2] + -7.567;
   1:L PR[91] R[100]mm/sec CNT100;
   1:  PR[91,1] = PR[90,1] + -39.122;
   1:  PR[91,2] = PR[90,2] + -8.820;
   1:L PR[91] R[100]mm/sec CNT100;
   1:  PR[91,1] = PR[90,1] + -38.825;
   1:  PR[91,2] = PR[90,2] + -9.370;
   1:L PR[91] R[100]mm/sec CNT100;
   1:  PR[91,1] = PR[90,1] + -37.086;
   1:  PR[91,2] = PR[90,2] + -12.138;
   1:L PR[91] R[100]mm/sec CNT100;
   1:  PR[91,1] = PR[90,1] + -36.794;
   1:  PR[91,2] = PR[90,2] + -12.551;
   1:L PR[91] R[100]mm/sec CNT100;
   1:  PR[91,1] = PR[90,1] + -36.056;
   1:  PR[91,2] = PR[90,2] + -13.368;
   1:L PR[91] R[100]mm/sec CNT100;
   1:  PR[91,1] = PR[90,1] + -33.732;
   1:  PR[91,2] = PR[90,2] + -15.700;
   1:L PR[91] R[100]mm/sec CNT100;
   1:  PR[91,1] = PR[90,1] + -32.622;
   1:  PR[91,2] = PR[90,2] + -16.492;
   1:L PR[91] R[100]mm/sec CNT100;
   1:  PR[91,1] = PR[90,1] + -30.086;
   1:  PR[91,2] = PR[90,2] + -18.111;
   1:L PR[91] R[100]mm/sec CNT100;
   1:  PR[91,1] = PR[90,1] + -28.459;
   1:  PR[91,2] = PR[90,2] + -18.807;
   1:L PR[91] R[100]mm/sec CNT100;
   1:  PR[91,1] = PR[90,1] + -25.985;
   1:  PR[91,2] = PR[90,2] + -19.712;
   1:L PR[91] R[100]mm/sec CNT100;
   1:  PR[91,1] = PR[90,1] + -23.769;
   1:  PR[91,2] = PR[90,2] + -20.140;
   1:L PR[91] R[100]mm/sec CNT100;
   1:  PR[91,1] = PR[90,1] + -21.612;
   1:  PR[91,2] = PR[90,2] + -20.432;
   1:L PR[91] R[100]mm/sec CNT100;
   1:  PR[91,1] = PR[90,1] + -18.812;
   1:  PR[91,2] = PR[90,2] + -20.365;
   1:L PR[91] R[100]mm/sec CNT100;
   1:  PR[91,1] = PR[90,1] + -17.167;
   1:  PR[91,2] = PR[90,2] + -20.229;
   1:L PR[91] R[100]mm/sec CNT100;
   1:  PR[91,1] = PR[90,1] + -13.883;
   1:  PR[91,2] = PR[90,2] + -19.427;
   1:L PR[91] R[100]mm/sec CNT100;
   1:  PR[91,1] = PR[90,1] + -12.850;
   1:  PR[91,2] = PR[90,2] + -19.107;
   1:L PR[91] R[100]mm/sec CNT100;
   1:  PR[91,1] = PR[90,1] + -9.308;
   1:  PR[91,2] = PR[90,2] + -17.354;
   1:L PR[91] R[100]mm/sec CNT100;
   1:  PR[91,1] = PR[90,1] + -8.864;
   1:  PR[91,2] = PR[90,2] + -17.098;
   1:L PR[91] R[100]mm/sec CNT100;
   1:  PR[91,1] = PR[90,1] + -5.397;
   1:  PR[91,2] = PR[90,2] + -14.278;
   1:L PR[91] R[100]mm/sec CNT100;
   1:  PR[91,1] = PR[90,1] + -3.913;
   1:  PR[91,2] = PR[90,2] + -12.363;
   1:L PR[91] R[100]mm/sec CNT100;
   1:  PR[91,1] = PR[90,1] + -2.510;
   1:  PR[91,2] = PR[90,2] + -10.642;
   1:L PR[91] R[100]mm/sec CNT100;
   1:  PR[91,1] = PR[90,1] + -2.507;
   1:  PR[91,2] = PR[90,2] + -10.636;
   1:L PR[91] R[100]mm/sec CNT100;
   1:  PR[91,1] = PR[90,1] + -0.715;
   1:  PR[91,2] = PR[90,2] + -6.857;
   1:L PR[91] R[100]mm/sec CNT100;
   1:  PR[91,1] = PR[90,1] + -0.610;
   1:  PR[91,2] = PR[90,2] + -6.577;
   1:L PR[91] R[100]mm/sec CNT100;
   1:  PR[91,1] = PR[90,1] + 0.216;
   1:  PR[91,2] = PR[90,2] + -3.257;
   1:L PR[91] R[100]mm/sec CNT100;
   1:  PR[91,1] = PR[90,1] + 3.385;
   1:  PR[91,2] = PR[90,2] + -3.299;
   1:L PR[91] R[100]mm/sec CNT100;
   1:  PR[91,1] = PR[90,1] + 4.076;
   1:  PR[91,2] = PR[90,2] + -6.422;
   1:L PR[91] R[100]mm/sec CNT100;
   1:  PR[91,1] = PR[90,1] + 4.773;
   1:  PR[91,2] = PR[90,2] + -8.090;
   1:L PR[91] R[100]mm/sec CNT100;
   1:  PR[91,1] = PR[90,1] + 5.666;
   1:  PR[91,2] = PR[90,2] + -10.320;
   1:L PR[91] R[100]mm/sec CNT100;
   1:  PR[91,1] = PR[90,1] + 6.034;
   1:  PR[91,2] = PR[90,2] + -11.054;
   1:L PR[91] R[100]mm/sec CNT100;
   1:  PR[91,1] = PR[90,1] + 8.671;
   1:  PR[91,2] = PR[90,2] + -14.460;
   1:L PR[91] R[100]mm/sec CNT100;
   1:  PR[91,1] = PR[90,1] + 8.949;
   1:  PR[91,2] = PR[90,2] + -14.860;
   1:L PR[91] R[100]mm/sec CNT100;
   1:  PR[91,1] = PR[90,1] + 9.487;
   1:  PR[91,2] = PR[90,2] + -15.427;
   1:L PR[91] R[100]mm/sec CNT100;
   1:  PR[91,1] = PR[90,1] + 13.137;
   1:  PR[91,2] = PR[90,2] + -18.194;
   1:L PR[91] R[100]mm/sec CNT100;
   1:  PR[91,1] = PR[90,1] + 13.723;
   1:  PR[91,2] = PR[90,2] + -18.559;
   1:L PR[91] R[100]mm/sec CNT100;
   1:  PR[91,1] = PR[90,1] + 18.095;
   1:  PR[91,2] = PR[90,2] + -20.344;
   1:L PR[91] R[100]mm/sec CNT100;
   1:  PR[91,1] = PR[90,1] + 18.615;
   1:  PR[91,2] = PR[90,2] + -20.509;
   1:L PR[91] R[100]mm/sec CNT100;
   1:  PR[91,1] = PR[90,1] + 23.451;
   1:  PR[91,2] = PR[90,2] + -21.128;
   1:L PR[91] R[100]mm/sec CNT100;
   1:  PR[91,1] = PR[90,1] + 23.842;
   1:  PR[91,2] = PR[90,2] + -21.151;
   1:L PR[91] R[100]mm/sec CNT100;
   1:  PR[91,1] = PR[90,1] + 28.822;
   1:  PR[91,2] = PR[90,2] + -20.487;
   1:L PR[91] R[100]mm/sec CNT100;
   1:  PR[91,1] = PR[90,1] + 29.059;
   1:  PR[91,2] = PR[90,2] + -20.442;
   1:L PR[91] R[100]mm/sec CNT100;
   1:  PR[91,1] = PR[90,1] + 33.829;
   1:  PR[91,2] = PR[90,2] + -18.475;
   1:L PR[91] R[100]mm/sec CNT100;
   1:  PR[91,1] = PR[90,1] + 33.923;
   1:  PR[91,2] = PR[90,2] + -18.431;
   1:L PR[91] R[100]mm/sec CNT100;
   1:  PR[91,1] = PR[90,1] + 38.131;
   1:  PR[91,2] = PR[90,2] + -15.244;
   1:L PR[91] R[100]mm/sec CNT100;
   1:  PR[91,1] = PR[90,1] + 38.658;
   1:  PR[91,2] = PR[90,2] + -14.617;
   1:L PR[91] R[100]mm/sec CNT100;
   1:  PR[91,1] = PR[90,1] + 42.705;
   1:  PR[91,2] = PR[90,2] + -9.418;
   1:L PR[91] R[100]mm/sec CNT100;
   1:  PR[91,1] = PR[90,1] + 47.189;
   1:  PR[91,2] = PR[90,2] + -14.100;
   1:L PR[91] R[100]mm/sec CNT100;
   1:  PR[91,1] = PR[90,1] + 47.481;
   1:  PR[91,2] = PR[90,2] + -14.437;
   1:L PR[91] R[100]mm/sec CNT100;
   1:  PR[91,1] = PR[90,1] + 50.974;
   1:  PR[91,2] = PR[90,2] + -16.993;
   1:L PR[91] R[100]mm/sec CNT100;
   1:  PR[91,1] = PR[90,1] + 52.879;
   1:  PR[91,2] = PR[90,2] + -18.168;
   1:L PR[91] R[100]mm/sec CNT100;
   1:  PR[91,1] = PR[90,1] + 55.023;
   1:  PR[91,2] = PR[90,2] + -19.106;
   1:L PR[91] R[100]mm/sec CNT100;
   1:  PR[91,1] = PR[90,1] + 59.619;
   1:  PR[91,2] = PR[90,2] + -20.650;
   1:L PR[91] R[100]mm/sec CNT100;
   1:  PR[91,1] = PR[90,1] + 59.641;
   1:  PR[91,2] = PR[90,2] + -20.654;
   1:L PR[91] R[100]mm/sec CNT100;
   1:  PR[91,1] = PR[90,1] + 60.098;
   1:  PR[91,2] = PR[90,2] + -20.706;
   1:L PR[91] R[100]mm/sec CNT100;
   1:  PR[91,1] = PR[90,1] + 64.803;
   1:  PR[91,2] = PR[90,2] + -21.406;
   1:L PR[91] R[100]mm/sec CNT100;
   1:  PR[91,1] = PR[90,1] + 66.209;
   1:  PR[91,2] = PR[90,2] + -21.457;
   1:L PR[91] R[100]mm/sec CNT100;
   1:  PR[91,1] = PR[90,1] + 69.518;
   1:  PR[91,2] = PR[90,2] + -21.226;
   1:L PR[91] R[100]mm/sec CNT100;
   1:  PR[91,1] = PR[90,1] + 72.304;
   1:  PR[91,2] = PR[90,2] + -20.762;
   1:L PR[91] R[100]mm/sec CNT100;
   1:  PR[91,1] = PR[90,1] + 73.960;
   1:  PR[91,2] = PR[90,2] + -20.276;
   1:L PR[91] R[100]mm/sec CNT100;
   1:  PR[91,1] = PR[90,1] + 77.569;
   1:  PR[91,2] = PR[90,2] + -18.895;
   1:L PR[91] R[100]mm/sec CNT100;
   1:  PR[91,1] = PR[90,1] + 78.035;
   1:  PR[91,2] = PR[90,2] + -18.638;
   1:L PR[91] R[100]mm/sec CNT100;
   1:  PR[91,1] = PR[90,1] + 81.794;
   1:  PR[91,2] = PR[90,2] + -16.221;
   1:L PR[91] R[100]mm/sec CNT100;
   1:  PR[91,1] = PR[90,1] + 84.969;
   1:  PR[91,2] = PR[90,2] + -12.992;
   1:L PR[91] R[100]mm/sec CNT100;
   1:  PR[91,1] = PR[90,1] + 87.334;
   1:  PR[91,2] = PR[90,2] + -9.214;
   1:L PR[91] R[100]mm/sec CNT100;
   1:  PR[91,1] = PR[90,1] + 88.789;
   1:  PR[91,2] = PR[90,2] + -5.064;
   1:L PR[91] R[100]mm/sec CNT100;
   1:  PR[91,1] = PR[90,1] + 89.281;
   1:  PR[91,2] = PR[90,2] + -0.729;
   1:L PR[91] R[100]mm/sec CNT100;
   1:  PR[91,1] = PR[90,1] + 88.789;
   1:  PR[91,2] = PR[90,2] + 3.606;
   1:L PR[91] R[100]mm/sec CNT100;
   1:  PR[91,1] = PR[90,1] + 87.334;
   1:  PR[91,2] = PR[90,2] + 7.755;
   1:L PR[91] R[100]mm/sec CNT100;
   1:  PR[91,1] = PR[90,1] + 84.969;
   1:  PR[91,2] = PR[90,2] + 11.533;
   1:L PR[91] R[100]mm/sec CNT100;
   1:  PR[91,1] = PR[90,1] + 81.794;
   1:  PR[91,2] = PR[90,2] + 14.762;
   1:L PR[91] R[100]mm/sec CNT100;
   1:  PR[91,1] = PR[90,1] + 78.035;
   1:  PR[91,2] = PR[90,2] + 17.179;
   1:L PR[91] R[100]mm/sec CNT100;
   1:  PR[91,1] = PR[90,1] + 77.569;
   1:  PR[91,2] = PR[90,2] + 17.436;
   1:L PR[91] R[100]mm/sec CNT100;
   1:  PR[91,1] = PR[90,1] + 73.960;
   1:  PR[91,2] = PR[90,2] + 18.817;
   1:L PR[91] R[100]mm/sec CNT100;
   1:  PR[91,1] = PR[90,1] + 72.304;
   1:  PR[91,2] = PR[90,2] + 19.303;
   1:L PR[91] R[100]mm/sec CNT100;
   1:  PR[91,1] = PR[90,1] + 69.518;
   1:  PR[91,2] = PR[90,2] + 19.767;
   1:L PR[91] R[100]mm/sec CNT100;
   1:  PR[91,1] = PR[90,1] + 66.210;
   1:  PR[91,2] = PR[90,2] + 19.998;
   1:L PR[91] R[100]mm/sec CNT100;
   1:  PR[91,1] = PR[90,1] + 64.803;
   1:  PR[91,2] = PR[90,2] + 19.947;
   1:L PR[91] R[100]mm/sec CNT100;
   1:  PR[91,1] = PR[90,1] + 60.098;
   1:  PR[91,2] = PR[90,2] + 19.247;
   1:L PR[91] R[100]mm/sec CNT100;
   1:  PR[91,1] = PR[90,1] + 59.643;
   1:  PR[91,2] = PR[90,2] + 19.196;
   1:L PR[91] R[100]mm/sec CNT100;
   1:  PR[91,1] = PR[90,1] + 59.618;
   1:  PR[91,2] = PR[90,2] + 19.191;
   1:L PR[91] R[100]mm/sec CNT100;
   1:  PR[91,1] = PR[90,1] + 55.003;
   1:  PR[91,2] = PR[90,2] + 17.641;
   1:L PR[91] R[100]mm/sec CNT100;
   1:  PR[91,1] = PR[90,1] + 52.828;
   1:  PR[91,2] = PR[90,2] + 16.681;
   1:L PR[91] R[100]mm/sec CNT100;
   1:  PR[91,1] = PR[90,1] + 50.931;
   1:  PR[91,2] = PR[90,2] + 15.513;
   1:L PR[91] R[100]mm/sec CNT100;
   1:  PR[91,1] = PR[90,1] + 47.400;
   1:  PR[91,2] = PR[90,2] + 12.904;
   1:L PR[91] R[100]mm/sec CNT100;
   1:  PR[91,1] = PR[90,1] + 47.207;
   1:  PR[91,2] = PR[90,2] + 12.680;
   1:L PR[91] R[100]mm/sec CNT100;
   1:  PR[91,1] = PR[90,1] + 42.713;
   1:  PR[91,2] = PR[90,2] + 7.937;
   1:L PR[91] R[100]mm/sec CNT100;
   1:  PR[91,1] = PR[90,1] + 38.150;
   1:  PR[91,2] = PR[90,2] + 13.761;
   1:L PR[91] R[100]mm/sec CNT100;
   1:  PR[91,1] = PR[90,1] + 38.071;
   1:  PR[91,2] = PR[90,2] + 13.839;
   1:L PR[91] R[100]mm/sec CNT100;
   1:  PR[91,1] = PR[90,1] + 33.925;
   1:  PR[91,2] = PR[90,2] + 16.974;
   1:L PR[91] R[100]mm/sec CNT100;
   1:  PR[91,1] = PR[90,1] + 33.918;
   1:  PR[91,2] = PR[90,2] + 16.979;
   1:L PR[91] R[100]mm/sec CNT100;
   1:  PR[91,1] = PR[90,1] + 33.792;
   1:  PR[91,2] = PR[90,2] + 17.038;
   1:L PR[91] R[100]mm/sec CNT100;
   1:  PR[91,1] = PR[90,1] + 29.024;
   1:  PR[91,2] = PR[90,2] + 18.992;
   1:L PR[91] R[100]mm/sec CNT100;
   1:  PR[91,1] = PR[90,1] + 28.786;
   1:  PR[91,2] = PR[90,2] + 19.038;
   1:L PR[91] R[100]mm/sec CNT100;
   1:  PR[91,1] = PR[90,1] + 23.812;
   1:  PR[91,2] = PR[90,2] + 19.692;
   1:L PR[91] R[100]mm/sec CNT100;
   1:  PR[91,1] = PR[90,1] + 23.421;
   1:  PR[91,2] = PR[90,2] + 19.670;
   1:L PR[91] R[100]mm/sec CNT100;
   1:  PR[91,1] = PR[90,1] + 18.592;
   1:  PR[91,2] = PR[90,2] + 19.044;
   1:L PR[91] R[100]mm/sec CNT100;
   1:  PR[91,1] = PR[90,1] + 18.072;
   1:  PR[91,2] = PR[90,2] + 18.880;
   1:L PR[91] R[100]mm/sec CNT100;
   1:  PR[91,1] = PR[90,1] + 13.707;
   1:  PR[91,2] = PR[90,2] + 17.092;
   1:L PR[91] R[100]mm/sec CNT100;
   1:  PR[91,1] = PR[90,1] + 13.121;
   1:  PR[91,2] = PR[90,2] + 16.727;
   1:L PR[91] R[100]mm/sec CNT100;
   1:  PR[91,1] = PR[90,1] + 9.478;
   1:  PR[91,2] = PR[90,2] + 13.959;
   1:L PR[91] R[100]mm/sec CNT100;
   1:  PR[91,1] = PR[90,1] + 8.904;
   1:  PR[91,2] = PR[90,2] + 13.356;
   1:L PR[91] R[100]mm/sec CNT100;
   1:  PR[91,1] = PR[90,1] + 6.144;
   1:  PR[91,2] = PR[90,2] + 9.789;
   1:L PR[91] R[100]mm/sec CNT100;
   1:  PR[91,1] = PR[90,1] + 6.104;
   1:  PR[91,2] = PR[90,2] + 9.727;
   1:L PR[91] R[100]mm/sec CNT100;
   1:  PR[91,1] = PR[90,1] + 5.769;
   1:  PR[91,2] = PR[90,2] + 9.085;
   1:L PR[91] R[100]mm/sec CNT100;
   1:  PR[91,1] = PR[90,1] + 4.383;
   1:  PR[91,2] = PR[90,2] + 5.768;
   1:L PR[91] R[100]mm/sec CNT100;
   1:  PR[91,1] = PR[90,1] + 4.103;
   1:  PR[91,2] = PR[90,2] + 5.061;
   1:L PR[91] R[100]mm/sec CNT100;
   1:  PR[91,1] = PR[90,1] + 3.380;
   1:  PR[91,2] = PR[90,2] + 1.835;
   1:L PR[91] R[100]mm/sec CNT100;
   1:  PR[91,1] = PR[90,1] + 0.218;
   1:  PR[91,2] = PR[90,2] + 1.796;
   1:L PR[91] R[100]mm/sec CNT100;
   1:  PR[91,1] = PR[90,1] + -0.605;
   1:  PR[91,2] = PR[90,2] + 5.086;
   1:L PR[91] R[100]mm/sec CNT100;
   1:  PR[91,1] = PR[90,1] + -2.193;
   1:  PR[91,2] = PR[90,2] + 8.477;
   1:L PR[91] R[100]mm/sec CNT100;
   1:  PR[91,1] = PR[90,1] + -2.509;
   1:  PR[91,2] = PR[90,2] + 9.179;
   1:L PR[91] R[100]mm/sec CNT100;
   1:  PR[91,1] = PR[90,1] + -3.914;
   1:  PR[91,2] = PR[90,2] + 10.905;
   1:L PR[91] R[100]mm/sec CNT100;
   1:  PR[91,1] = PR[90,1] + -5.385;
   1:  PR[91,2] = PR[90,2] + 12.808;
   1:L PR[91] R[100]mm/sec CNT100;
   1:  PR[91,1] = PR[90,1] + -8.852;
   1:  PR[91,2] = PR[90,2] + 15.632;
   1:L PR[91] R[100]mm/sec CNT100;
   1:  PR[91,1] = PR[90,1] + -9.296;
   1:  PR[91,2] = PR[90,2] + 15.887;
   1:L PR[91] R[100]mm/sec CNT100;
   1:  PR[91,1] = PR[90,1] + -12.840;
   1:  PR[91,2] = PR[90,2] + 17.644;
   1:L PR[91] R[100]mm/sec CNT100;
   1:  PR[91,1] = PR[90,1] + -13.871;
   1:  PR[91,2] = PR[90,2] + 17.964;
   1:L PR[91] R[100]mm/sec CNT100;
   1:  PR[91,1] = PR[90,1] + -17.158;
   1:  PR[91,2] = PR[90,2] + 18.769;
   1:L PR[91] R[100]mm/sec CNT100;
   1:  PR[91,1] = PR[90,1] + -18.802;
   1:  PR[91,2] = PR[90,2] + 18.905;
   1:L PR[91] R[100]mm/sec CNT100;
   1:  PR[91,1] = PR[90,1] + -21.605;
   1:  PR[91,2] = PR[90,2] + 18.974;
   1:L PR[91] R[100]mm/sec CNT100;
   1:  PR[91,1] = PR[90,1] + -23.761;
   1:  PR[91,2] = PR[90,2] + 18.682;
   1:L PR[91] R[100]mm/sec CNT100;
   1:  PR[91,1] = PR[90,1] + -25.979;
   1:  PR[91,2] = PR[90,2] + 18.255;
   1:L PR[91] R[100]mm/sec CNT100;
   1:  PR[91,1] = PR[90,1] + -28.453;
   1:  PR[91,2] = PR[90,2] + 17.350;
   1:L PR[91] R[100]mm/sec CNT100;
   1:  PR[91,1] = PR[90,1] + -30.082;
   1:  PR[91,2] = PR[90,2] + 16.654;
   1:L PR[91] R[100]mm/sec CNT100;
   1:  PR[91,1] = PR[90,1] + -32.618;
   1:  PR[91,2] = PR[90,2] + 15.035;
   1:L PR[91] R[100]mm/sec CNT100;
   1:  PR[91,1] = PR[90,1] + -33.730;
   1:  PR[91,2] = PR[90,2] + 14.244;
   1:L PR[91] R[100]mm/sec CNT100;
   1:  PR[91,1] = PR[90,1] + -36.054;
   1:  PR[91,2] = PR[90,2] + 11.911;
   1:L PR[91] R[100]mm/sec CNT100;
   1:  PR[91,1] = PR[90,1] + -36.756;
   1:  PR[91,2] = PR[90,2] + 11.135;
   1:L PR[91] R[100]mm/sec CNT100;
   1:  PR[91,1] = PR[90,1] + -38.708;
   1:  PR[91,2] = PR[90,2] + 8.037;
   1:L PR[91] R[100]mm/sec CNT100;
   1:  PR[91,1] = PR[90,1] + -38.832;
   1:  PR[91,2] = PR[90,2] + 7.886;
   1:L PR[91] R[100]mm/sec CNT100;
   1:  PR[91,1] = PR[90,1] + -38.946;
   1:  PR[91,2] = PR[90,2] + 7.712;
   1:L PR[91] R[100]mm/sec CNT100;
   1:  PR[91,1] = PR[90,1] + -39.077;
   1:  PR[91,2] = PR[90,2] + 7.458;
   1:L PR[91] R[100]mm/sec CNT100;
   1:  PR[91,1] = PR[90,1] + -40.128;
   1:  PR[91,2] = PR[90,2] + 4.457;
   1:L PR[91] R[100]mm/sec CNT100;
   1:  PR[91,1] = PR[90,1] + -40.199;
   1:  PR[91,2] = PR[90,2] + 4.341;
   1:L PR[91] R[100]mm/sec CNT100TB   .50sec,CALL END_PUD;
   1:  PR[92] = PR[91];
   1:  PR[92,3] = PR[92,3] + 20;
   1:J PR[92] 10% FINE;
   1:  PR[91] = PR[90];
   1:  PR[91,1] = PR[90,1] + -65.992;
   1:  PR[91,2] = PR[90,2] + 18.957;
   1:  PR[91,3] = PR[90,3] + 40.495;
   1:  PR[92] = PR[91];
   1:  PR[92,3] = PR[92,3] + 20;
   1:J PR[92] 10% FINE;
   1:L PR[91] R[100]mm/sec CNT100;
   1:  CALL LASER_DRAHT_START;
   1:  PR[91,1] = PR[90,1] + -70.510;
   1:  PR[91,2] = PR[90,2] + 18.756;
   1:L PR[91] R[100]mm/sec CNT100;
   1:  PR[91,1] = PR[90,1] + -72.599;
   1:  PR[91,2] = PR[90,2] + 18.270;
   1:  PR[91,3] = PR[90,3] + 39.207;
   1:L PR[91] R[100]mm/sec CNT100;
   1:  PR[91,1] = PR[90,1] + -74.831;
   1:  PR[91,2] = PR[90,2] + 17.729;
   1:  PR[91,3] = PR[90,3] + 39.213;
   1:L PR[91] R[100]mm/sec CNT100;
   1:  PR[91,1] = PR[90,1] + -78.808;
   1:  PR[91,2] = PR[90,2] + 15.932;
   1:  PR[91,3] = PR[90,3] + 39.219;
   1:L PR[91] R[100]mm/sec CNT100;
   1:  PR[91,1] = PR[90,1] + -82.272;
   1:  PR[91,2] = PR[90,2] + 13.461;
   1:  PR[91,3] = PR[90,3] + 39.231;
   1:L PR[91] R[100]mm/sec CNT100;
   1:  PR[91,1] = PR[90,1] + -85.098;
   1:  PR[91,2] = PR[90,2] + 10.424;
   1:  PR[91,3] = PR[90,3] + 39.243;
   1:L PR[91] R[100]mm/sec CNT100;
   1:  PR[91,1] = PR[90,1] + -85.488;
   1:  PR[91,2] = PR[90,2] + 9.776;
   1:  PR[91,3] = PR[90,3] + 39.254;
   1:L PR[91] R[100]mm/sec CNT100;
   1:  PR[91,1] = PR[90,1] + -87.119;
   1:  PR[91,2] = PR[90,2] + 6.978;
   1:  PR[91,3] = PR[90,3] + 39.256;
   1:L PR[91] R[100]mm/sec CNT100;
   1:  PR[91,1] = PR[90,1] + -88.368;
   1:  PR[91,2] = PR[90,2] + 3.180;
   1:  PR[91,3] = PR[90,3] + 39.265;
   1:L PR[91] R[100]mm/sec CNT100;
   1:  PR[91,1] = PR[90,1] + -88.408;
   1:  PR[91,2] = PR[90,2] + 2.869;
   1:  PR[91,3] = PR[90,3] + 39.276;
   1:L PR[91] R[100]mm/sec CNT100;
   1:  PR[91,1] = PR[90,1] + -88.794;
   1:  PR[91,2] = PR[90,2] + -0.728;
   1:  PR[91,3] = PR[90,3] + 39.277;
   1:L PR[91] R[100]mm/sec CNT100;
   1:  PR[91,1] = PR[90,1] + -88.766;
   1:  PR[91,2] = PR[90,2] + -0.984;
   1:  PR[91,3] = PR[90,3] + 39.286;
   1:L PR[91] R[100]mm/sec CNT100;
   1:  PR[91,1] = PR[90,1] + -88.520;
   1:  PR[91,2] = PR[90,2] + -2.078;
   1:  PR[91,3] = PR[90,3] + 39.287;
   1:L PR[91] R[100]mm/sec CNT100;
   1:  PR[91,1] = PR[90,1] + -88.244;
   1:  PR[91,2] = PR[90,2] + -4.663;
   1:  PR[91,3] = PR[90,3] + 39.290;
   1:L PR[91] R[100]mm/sec CNT100;
   1:  PR[91,1] = PR[90,1] + -86.993;
   1:  PR[91,2] = PR[90,2] + -8.441;
   1:  PR[91,3] = PR[90,3] + 39.297;
   1:L PR[91] R[100]mm/sec CNT100;
   1:  PR[91,1] = PR[90,1] + -84.954;
   1:  PR[91,2] = PR[90,2] + -11.914;
   1:  PR[91,3] = PR[90,3] + 39.308;
   1:L PR[91] R[100]mm/sec CNT100;
   1:  PR[91,1] = PR[90,1] + -82.204;
   1:  PR[91,2] = PR[90,2] + -14.942;
   1:  PR[91,3] = PR[90,3] + 39.319;
   1:L PR[91] R[100]mm/sec CNT100;
   1:  PR[91,1] = PR[90,1] + -78.842;
   1:  PR[91,2] = PR[90,2] + -17.393;
   1:  PR[91,3] = PR[90,3] + 39.330;
   1:L PR[91] R[100]mm/sec CNT100;
   1:  PR[91,1] = PR[90,1] + -76.437;
   1:  PR[91,2] = PR[90,2] + -18.498;
   1:  PR[91,3] = PR[90,3] + 39.341;
   1:L PR[91] R[100]mm/sec CNT100;
   1:  PR[91,1] = PR[90,1] + -74.938;
   1:  PR[91,2] = PR[90,2] + -19.169;
   1:  PR[91,3] = PR[90,3] + 39.349;
   1:L PR[91] R[100]mm/sec CNT100;
   1:  PR[91,1] = PR[90,1] + -71.259;
   1:  PR[91,2] = PR[90,2] + -20.025;
   1:  PR[91,3] = PR[90,3] + 39.353;
   1:L PR[91] R[100]mm/sec CNT100;
   1:  PR[91,1] = PR[90,1] + -70.510;
   1:  PR[91,2] = PR[90,2] + -20.211;
   1:  PR[91,3] = PR[90,3] + 39.363;
   1:L PR[91] R[100]mm/sec CNT100;
   1:  PR[91,1] = PR[90,1] + -67.495;
   1:  PR[91,2] = PR[90,2] + -20.334;
   1:  PR[91,3] = PR[90,3] + 39.365;
   1:L PR[91] R[100]mm/sec CNT100;
   1:  PR[91,1] = PR[90,1] + -65.902;
   1:  PR[91,2] = PR[90,2] + -20.425;
   1:  PR[91,3] = PR[90,3] + 39.374;
   1:L PR[91] R[100]mm/sec CNT100;
   1:  PR[91,1] = PR[90,1] + -63.771;
   1:  PR[91,2] = PR[90,2] + -20.108;
   1:  PR[91,3] = PR[90,3] + 39.378;
   1:L PR[91] R[100]mm/sec CNT100;
   1:  PR[91,1] = PR[90,1] + -61.287;
   1:  PR[91,2] = PR[90,2] + -19.782;
   1:  PR[91,3] = PR[90,3] + 39.384;
   1:L PR[91] R[100]mm/sec CNT100;
   1:  PR[91,1] = PR[90,1] + -60.163;
   1:  PR[91,2] = PR[90,2] + -19.383;
   1:  PR[91,3] = PR[90,3] + 39.391;
   1:L PR[91] R[100]mm/sec CNT100;
   1:  PR[91,1] = PR[90,1] + -56.854;
   1:  PR[91,2] = PR[90,2] + -18.276;
   1:  PR[91,3] = PR[90,3] + 39.394;
   1:L PR[91] R[100]mm/sec CNT100;
   1:  PR[91,1] = PR[90,1] + -55.345;
   1:  PR[91,2] = PR[90,2] + -17.399;
   1:  PR[91,3] = PR[90,3] + 39.403;
   1:L PR[91] R[100]mm/sec CNT100;
   1:  PR[91,1] = PR[90,1] + -52.784;
   1:  PR[91,2] = PR[90,2] + -16.071;
   1:  PR[91,3] = PR[90,3] + 39.408;
   1:L PR[91] R[100]mm/sec CNT100;
   1:  PR[91,1] = PR[90,1] + -52.031;
   1:  PR[91,2] = PR[90,2] + -15.552;
   1:  PR[91,3] = PR[90,3] + 39.416;
   1:L PR[91] R[100]mm/sec CNT100;
   1:  PR[91,1] = PR[90,1] + -49.353;
   1:  PR[91,2] = PR[90,2] + -13.360;
   1:  PR[91,3] = PR[90,3] + 39.418;
   1:L PR[91] R[100]mm/sec CNT100;
   1:  PR[91,1] = PR[90,1] + -47.673;
   1:  PR[91,2] = PR[90,2] + -11.503;
   1:  PR[91,3] = PR[90,3] + 39.428;
   1:L PR[91] R[100]mm/sec CNT100;
   1:  PR[91,1] = PR[90,1] + -46.502;
   1:  PR[91,2] = PR[90,2] + -9.984;
   1:  PR[91,3] = PR[90,3] + 39.435;
   1:L PR[91] R[100]mm/sec CNT100;
   1:  PR[91,1] = PR[90,1] + -44.819;
   1:  PR[91,2] = PR[90,2] + -6.737;
   1:  PR[91,3] = PR[90,3] + 39.440;
   1:L PR[91] R[100]mm/sec CNT100;
   1:  PR[91,1] = PR[90,1] + -44.494;
   1:  PR[91,2] = PR[90,2] + -5.982;
   1:  PR[91,3] = PR[90,3] + 39.450;
   1:L PR[91] R[100]mm/sec CNT100;
   1:  PR[91,1] = PR[90,1] + -43.886;
   1:  PR[91,2] = PR[90,2] + -3.116;
   1:  PR[91,3] = PR[90,3] + 39.452;
   1:L PR[91] R[100]mm/sec CNT100;
   1:  PR[91,1] = PR[90,1] + -40.672;
   1:  PR[91,2] = PR[90,2] + -3.090;
   1:  PR[91,3] = PR[90,3] + 39.460;
   1:L PR[91] R[100]mm/sec CNT100;
   1:  PR[91,1] = PR[90,1] + -40.009;
   1:  PR[91,2] = PR[90,2] + -5.989;
   1:  PR[91,3] = PR[90,3] + 39.469;
   1:L PR[91] R[100]mm/sec CNT100;
   1:  PR[91,1] = PR[90,1] + -39.713;
   1:  PR[91,2] = PR[90,2] + -6.837;
   1:  PR[91,3] = PR[90,3] + 39.477;
   1:L PR[91] R[100]mm/sec CNT100;
   1:  PR[91,1] = PR[90,1] + -38.974;
   1:  PR[91,2] = PR[90,2] + -8.740;
   1:  PR[91,3] = PR[90,3] + 39.479;
   1:L PR[91] R[100]mm/sec CNT100;
   1:  PR[91,1] = PR[90,1] + -38.498;
   1:  PR[91,2] = PR[90,2] + -9.622;
   1:  PR[91,3] = PR[90,3] + 39.485;
   1:L PR[91] R[100]mm/sec CNT100;
   1:  PR[91,1] = PR[90,1] + -37.059;
   1:  PR[91,2] = PR[90,2] + -11.912;
   1:  PR[91,3] = PR[90,3] + 39.487;
   1:L PR[91] R[100]mm/sec CNT100;
   1:  PR[91,1] = PR[90,1] + -36.612;
   1:  PR[91,2] = PR[90,2] + -12.544;
   1:  PR[91,3] = PR[90,3] + 39.495;
   1:L PR[91] R[100]mm/sec CNT100;
   1:  PR[91,1] = PR[90,1] + -35.538;
   1:  PR[91,2] = PR[90,2] + -13.733;
   1:  PR[91,3] = PR[90,3] + 39.497;
   1:L PR[91] R[100]mm/sec CNT100;
   1:  PR[91,1] = PR[90,1] + -33.554;
   1:  PR[91,2] = PR[90,2] + -15.725;
   1:  PR[91,3] = PR[90,3] + 39.501;
   1:L PR[91] R[100]mm/sec CNT100;
   1:  PR[91,1] = PR[90,1] + -32.019;
   1:  PR[91,2] = PR[90,2] + -16.819;
   1:  PR[91,3] = PR[90,3] + 39.509;
   1:L PR[91] R[100]mm/sec CNT100;
   1:  PR[91,1] = PR[90,1] + -29.908;
   1:  PR[91,2] = PR[90,2] + -18.167;
   1:  PR[91,3] = PR[90,3] + 39.514;
   1:L PR[91] R[100]mm/sec CNT100;
   1:  PR[91,1] = PR[90,1] + -27.776;
   1:  PR[91,2] = PR[90,2] + -19.079;
   1:  PR[91,3] = PR[90,3] + 39.521;
   1:L PR[91] R[100]mm/sec CNT100;
   1:  PR[91,1] = PR[90,1] + -25.799;
   1:  PR[91,2] = PR[90,2] + -19.802;
   1:  PR[91,3] = PR[90,3] + 39.527;
   1:L PR[91] R[100]mm/sec CNT100;
   1:  PR[91,1] = PR[90,1] + -23.017;
   1:  PR[91,2] = PR[90,2] + -20.339;
   1:  PR[91,3] = PR[90,3] + 39.533;
   1:L PR[91] R[100]mm/sec CNT100;
   1:  PR[91,1] = PR[90,1] + -21.413;
   1:  PR[91,2] = PR[90,2] + -20.557;
   1:  PR[91,3] = PR[90,3] + 39.541;
   1:L PR[91] R[100]mm/sec CNT100;
   1:  PR[91,1] = PR[90,1] + -18.007;
   1:  PR[91,2] = PR[90,2] + -20.475;
   1:  PR[91,3] = PR[90,3] + 39.545;
   1:L PR[91] R[100]mm/sec CNT100;
   1:  PR[91,1] = PR[90,1] + -16.945;
   1:  PR[91,2] = PR[90,2] + -20.387;
   1:  PR[91,3] = PR[90,3] + 39.554;
   1:L PR[91] R[100]mm/sec CNT100;
   1:  PR[91,1] = PR[90,1] + -13.047;
   1:  PR[91,2] = PR[90,2] + -19.435;
   1:  PR[91,3] = PR[90,3] + 39.557;
   1:L PR[91] R[100]mm/sec CNT100;
   1:  PR[91,1] = PR[90,1] + -12.597;
   1:  PR[91,2] = PR[90,2] + -19.296;
   1:  PR[91,3] = PR[90,3] + 39.568;
   1:L PR[91] R[100]mm/sec CNT100;
   1:  PR[91,1] = PR[90,1] + -8.520;
   1:  PR[91,2] = PR[90,2] + -17.271;
   1:  PR[91,3] = PR[90,3] + 39.569;
   1:L PR[91] R[100]mm/sec CNT100;
   1:  PR[91,1] = PR[90,1] + -7.905;
   1:  PR[91,2] = PR[90,2] + -16.771;
   1:  PR[91,3] = PR[90,3] + 39.582;
   1:L PR[91] R[100]mm/sec CNT100;
   1:  PR[91,1] = PR[90,1] + -4.834;
   1:  PR[91,2] = PR[90,2] + -14.411;
   1:  PR[91,3] = PR[90,3] + 39.584;
   1:L PR[91] R[100]mm/sec CNT100;
   1:  PR[91,1] = PR[90,1] + -4.616;
   1:  PR[91,2] = PR[90,2] + -14.178;
   1:  PR[91,3] = PR[90,3] + 39.594;
   1:L PR[91] R[100]mm/sec CNT100;
   1:  PR[91,1] = PR[90,1] + -1.952;
   1:  PR[91,2] = PR[90,2] + -10.910;
   1:  PR[91,3] = PR[90,3] + 39.595;
   1:L PR[91] R[100]mm/sec CNT100;
   1:  PR[91,1] = PR[90,1] + -1.574;
   1:  PR[91,2] = PR[90,2] + -10.195;
   1:  PR[91,3] = PR[90,3] + 39.607;
   1:L PR[91] R[100]mm/sec CNT100;
   1:  PR[91,1] = PR[90,1] + -0.351;
   1:  PR[91,2] = PR[90,2] + -7.616;
   1:  PR[91,3] = PR[90,3] + 39.609;
   1:L PR[91] R[100]mm/sec CNT100;
   1:  PR[91,1] = PR[90,1] + -0.010;
   1:  PR[91,2] = PR[90,2] + -6.708;
   1:  PR[91,3] = PR[90,3] + 39.617;
   1:L PR[91] R[100]mm/sec CNT100;
   1:  PR[91,1] = PR[90,1] + 0.373;
   1:  PR[91,2] = PR[90,2] + -5.172;
   1:  PR[91,3] = PR[90,3] + 39.619;
   1:L PR[91] R[100]mm/sec CNT100;
   1:  PR[91,1] = PR[90,1] + 3.542;
   1:  PR[91,2] = PR[90,2] + -5.213;
   1:  PR[91,3] = PR[90,3] + 39.624;
   1:L PR[91] R[100]mm/sec CNT100;
   1:  PR[91,1] = PR[90,1] + 3.871;
   1:  PR[91,2] = PR[90,2] + -6.703;
   1:  PR[91,3] = PR[90,3] + 39.632;
   1:L PR[91] R[100]mm/sec CNT100;
   1:  PR[91,1] = PR[90,1] + 5.193;
   1:  PR[91,2] = PR[90,2] + -9.999;
   1:  PR[91,3] = PR[90,3] + 39.636;
   1:L PR[91] R[100]mm/sec CNT100;
   1:  PR[91,1] = PR[90,1] + 5.803;
   1:  PR[91,2] = PR[90,2] + -11.215;
   1:  PR[91,3] = PR[90,3] + 39.646;
   1:L PR[91] R[100]mm/sec CNT100;
   1:  PR[91,1] = PR[90,1] + 8.008;
   1:  PR[91,2] = PR[90,2] + -14.064;
   1:  PR[91,3] = PR[90,3] + 39.650;
   1:L PR[91] R[100]mm/sec CNT100;
   1:  PR[91,1] = PR[90,1] + 8.465;
   1:  PR[91,2] = PR[90,2] + -14.721;
   1:  PR[91,3] = PR[90,3] + 39.659;
   1:L PR[91] R[100]mm/sec CNT100;
   1:  PR[91,1] = PR[90,1] + 9.404;
   1:  PR[91,2] = PR[90,2] + -15.711;
   1:  PR[91,3] = PR[90,3] + 39.662;
   1:L PR[91] R[100]mm/sec CNT100;
   1:  PR[91,1] = PR[90,1] + 12.621;
   1:  PR[91,2] = PR[90,2] + -18.150;
   1:  PR[91,3] = PR[90,3] + 39.665;
   1:L PR[91] R[100]mm/sec CNT100;
   1:  PR[91,1] = PR[90,1] + 13.690;
   1:  PR[91,2] = PR[90,2] + -18.816;
   1:  PR[91,3] = PR[90,3] + 39.676;
   1:L PR[91] R[100]mm/sec CNT100;
   1:  PR[91,1] = PR[90,1] + 17.565;
   1:  PR[91,2] = PR[90,2] + -20.398;
   1:  PR[91,3] = PR[90,3] + 39.680;
   1:L PR[91] R[100]mm/sec CNT100;
   1:  PR[91,1] = PR[90,1] + 18.622;
   1:  PR[91,2] = PR[90,2] + -20.733;
   1:  PR[91,3] = PR[90,3] + 39.691;
   1:L PR[91] R[100]mm/sec CNT100;
   1:  PR[91,1] = PR[90,1] + 22.930;
   1:  PR[91,2] = PR[90,2] + -21.284;
   1:  PR[91,3] = PR[90,3] + 39.694;
   1:L PR[91] R[100]mm/sec CNT100;
   1:  PR[91,1] = PR[90,1] + 23.878;
   1:  PR[91,2] = PR[90,2] + -21.339;
   1:  PR[91,3] = PR[90,3] + 39.706;
   1:L PR[91] R[100]mm/sec CNT100;
   1:  PR[91,1] = PR[90,1] + 28.337;
   1:  PR[91,2] = PR[90,2] + -20.745;
   1:  PR[91,3] = PR[90,3] + 39.708;
   1:L PR[91] R[100]mm/sec CNT100;
   1:  PR[91,1] = PR[90,1] + 29.114;
   1:  PR[91,2] = PR[90,2] + -20.594;
   1:  PR[91,3] = PR[90,3] + 39.721;
   1:L PR[91] R[100]mm/sec CNT100;
   1:  PR[91,1] = PR[90,1] + 33.406;
   1:  PR[91,2] = PR[90,2] + -18.825;
   1:  PR[91,3] = PR[90,3] + 39.723;
   1:L PR[91] R[100]mm/sec CNT100;
   1:  PR[91,1] = PR[90,1] + 33.989;
   1:  PR[91,2] = PR[90,2] + -18.551;
   1:  PR[91,3] = PR[90,3] + 39.735;
   1:L PR[91] R[100]mm/sec CNT100;
   1:  PR[91,1] = PR[90,1] + 37.880;
   1:  PR[91,2] = PR[90,2] + -15.598;
   1:  PR[91,3] = PR[90,3] + 39.737;
   1:L PR[91] R[100]mm/sec CNT100;
   1:  PR[91,1] = PR[90,1] + 37.983;
   1:  PR[91,2] = PR[90,2] + -15.533;
   1:  PR[91,3] = PR[90,3] + 39.750;
   1:L PR[91] R[100]mm/sec CNT100;
   1:  PR[91,1] = PR[90,1] + 38.302;
   1:  PR[91,2] = PR[90,2] + -15.236;
   1:  PR[91,3] = PR[90,3] + 39.751;
   1:L PR[91] R[100]mm/sec CNT100;
   1:  PR[91,1] = PR[90,1] + 38.533;
   1:  PR[91,2] = PR[90,2] + -14.984;
   1:  PR[91,3] = PR[90,3] + 39.752;
   1:L PR[91] R[100]mm/sec CNT100;
   1:  PR[91,1] = PR[90,1] + 40.180;
   1:  PR[91,2] = PR[90,2] + -12.996;
   1:  PR[91,3] = PR[90,3] + 39.753;
   1:L PR[91] R[100]mm/sec CNT100;
   1:  PR[91,1] = PR[90,1] + 42.121;
   1:  PR[91,2] = PR[90,2] + -10.502;
   1:  PR[91,3] = PR[90,3] + 39.760;
   1:L PR[91] R[100]mm/sec CNT100;
   1:  PR[91,1] = PR[90,1] + 44.418;
   1:  PR[91,2] = PR[90,2] + -12.906;
   1:  PR[91,3] = PR[90,3] + 39.768;
   1:L PR[91] R[100]mm/sec CNT100;
   1:  PR[91,1] = PR[90,1] + 45.836;
   1:  PR[91,2] = PR[90,2] + -14.345;
   1:  PR[91,3] = PR[90,3] + 39.778;
   1:L PR[91] R[100]mm/sec CNT100;
   1:  PR[91,1] = PR[90,1] + 46.719;
   1:  PR[91,2] = PR[90,2] + -14.975;
   1:  PR[91,3] = PR[90,3] + 39.783;
   1:L PR[91] R[100]mm/sec CNT100;
   1:  PR[91,1] = PR[90,1] + 48.779;
   1:  PR[91,2] = PR[90,2] + -16.323;
   1:  PR[91,3] = PR[90,3] + 39.786;
   1:L PR[91] R[100]mm/sec CNT100;
   1:  PR[91,1] = PR[90,1] + 50.613;
   1:  PR[91,2] = PR[90,2] + -17.665;
   1:  PR[91,3] = PR[90,3] + 39.793;
   1:L PR[91] R[100]mm/sec CNT100;
   1:  PR[91,1] = PR[90,1] + 51.361;
   1:  PR[91,2] = PR[90,2] + -18.127;
   1:  PR[91,3] = PR[90,3] + 39.799;
   1:L PR[91] R[100]mm/sec CNT100;
   1:  PR[91,1] = PR[90,1] + 54.713;
   1:  PR[91,2] = PR[90,2] + -19.592;
   1:  PR[91,3] = PR[90,3] + 39.801;
   1:L PR[91] R[100]mm/sec CNT100;
   1:  PR[91,1] = PR[90,1] + 58.060;
   1:  PR[91,2] = PR[90,2] + -20.717;
   1:  PR[91,3] = PR[90,3] + 39.811;
   1:L PR[91] R[100]mm/sec CNT100;
   1:  PR[91,1] = PR[90,1] + 59.336;
   1:  PR[91,2] = PR[90,2] + -20.988;
   1:  PR[91,3] = PR[90,3] + 39.821;
   1:L PR[91] R[100]mm/sec CNT100;
   1:  PR[91,1] = PR[90,1] + 62.627;
   1:  PR[91,2] = PR[90,2] + -21.359;
   1:  PR[91,3] = PR[90,3] + 39.824;
   1:L PR[91] R[100]mm/sec CNT100;
   1:  PR[91,1] = PR[90,1] + 64.586;
   1:  PR[91,2] = PR[90,2] + -21.650;
   1:  PR[91,3] = PR[90,3] + 39.833;
   1:L PR[91] R[100]mm/sec CNT100;
   1:  PR[91,1] = PR[90,1] + 65.060;
   1:  PR[91,2] = PR[90,2] + -21.667;
   1:  PR[91,3] = PR[90,3] + 39.839;
   1:L PR[91] R[100]mm/sec CNT100;
   1:  PR[91,1] = PR[90,1] + 69.373;
   1:  PR[91,2] = PR[90,2] + -21.367;
   1:  PR[91,3] = PR[90,3] + 39.840;
   1:L PR[91] R[100]mm/sec CNT100;
   1:  PR[91,1] = PR[90,1] + 71.350;
   1:  PR[91,2] = PR[90,2] + -21.037;
   1:  PR[91,3] = PR[90,3] + 39.852;
   1:L PR[91] R[100]mm/sec CNT100;
   1:  PR[91,1] = PR[90,1] + 73.854;
   1:  PR[91,2] = PR[90,2] + -20.302;
   1:  PR[91,3] = PR[90,3] + 39.857;
   1:L PR[91] R[100]mm/sec CNT100;
   1:  PR[91,1] = PR[90,1] + 76.784;
   1:  PR[91,2] = PR[90,2] + -19.181;
   1:  PR[91,3] = PR[90,3] + 39.864;
   1:L PR[91] R[100]mm/sec CNT100;
   1:  PR[91,1] = PR[90,1] + 77.938;
   1:  PR[91,2] = PR[90,2] + -18.543;
   1:  PR[91,3] = PR[90,3] + 39.873;
   1:L PR[91] R[100]mm/sec CNT100;
   1:  PR[91,1] = PR[90,1] + 81.256;
   1:  PR[91,2] = PR[90,2] + -16.417;
   1:  PR[91,3] = PR[90,3] + 39.876;
   1:L PR[91] R[100]mm/sec CNT100;
   1:  PR[91,1] = PR[90,1] + 81.539;
   1:  PR[91,2] = PR[90,2] + -16.165;
   1:  PR[91,3] = PR[90,3] + 39.887;
   1:L PR[91] R[100]mm/sec CNT100;
   1:  PR[91,1] = PR[90,1] + 84.672;
   1:  PR[91,2] = PR[90,2] + -13.054;
   1:  PR[91,3] = PR[90,3] + 39.888;
   1:L PR[91] R[100]mm/sec CNT100;
   1:  PR[91,1] = PR[90,1] + 87.040;
   1:  PR[91,2] = PR[90,2] + -9.263;
   1:  PR[91,3] = PR[90,3] + 39.900;
   1:L PR[91] R[100]mm/sec CNT100;
   1:  PR[91,1] = PR[90,1] + 88.500;
   1:  PR[91,2] = PR[90,2] + -5.089;
   1:  PR[91,3] = PR[90,3] + 39.912;
   1:L PR[91] R[100]mm/sec CNT100;
   1:  PR[91,1] = PR[90,1] + 88.994;
   1:  PR[91,2] = PR[90,2] + -0.729;
   1:  PR[91,3] = PR[90,3] + 39.924;
   1:L PR[91] R[100]mm/sec CNT100;
   1:  PR[91,1] = PR[90,1] + 88.500;
   1:  PR[91,2] = PR[90,2] + 3.631;
   1:  PR[91,3] = PR[90,3] + 39.936;
   1:L PR[91] R[100]mm/sec CNT100;
   1:  PR[91,1] = PR[90,1] + 87.040;
   1:  PR[91,2] = PR[90,2] + 7.804;
   1:  PR[91,3] = PR[90,3] + 39.948;
   1:L PR[91] R[100]mm/sec CNT100;
   1:  PR[91,1] = PR[90,1] + 84.672;
   1:  PR[91,2] = PR[90,2] + 11.595;
   1:  PR[91,3] = PR[90,3] + 39.960;
   1:L PR[91] R[100]mm/sec CNT100;
   1:  PR[91,1] = PR[90,1] + 81.539;
   1:  PR[91,2] = PR[90,2] + 14.706;
   1:  PR[91,3] = PR[90,3] + 39.972;
   1:L PR[91] R[100]mm/sec CNT100;
   1:  PR[91,1] = PR[90,1] + 81.256;
   1:  PR[91,2] = PR[90,2] + 14.958;
   1:  PR[91,3] = PR[90,3] + 39.984;
   1:L PR[91] R[100]mm/sec CNT100;
   1:  PR[91,1] = PR[90,1] + 77.939;
   1:  PR[91,2] = PR[90,2] + 17.085;
   1:  PR[91,3] = PR[90,3] + 39.985;
   1:L PR[91] R[100]mm/sec CNT100;
   1:  PR[91,1] = PR[90,1] + 76.784;
   1:  PR[91,2] = PR[90,2] + 17.723;
   1:  PR[91,3] = PR[90,3] + 39.996;
   1:L PR[91] R[100]mm/sec CNT100;
   1:  PR[91,1] = PR[90,1] + 73.855;
   1:  PR[91,2] = PR[90,2] + 18.843;
   1:  PR[91,3] = PR[90,3] + 40.000;
   1:L PR[91] R[100]mm/sec CNT100;
   1:  PR[91,1] = PR[90,1] + 71.351;
   1:  PR[91,2] = PR[90,2] + 19.578;
   1:  PR[91,3] = PR[90,3] + 40.008;
   1:L PR[91] R[100]mm/sec CNT100;
   1:  PR[91,1] = PR[90,1] + 69.373;
   1:  PR[91,2] = PR[90,2] + 19.908;
   1:  PR[91,3] = PR[90,3] + 40.015;
   1:L PR[91] R[100]mm/sec CNT100;
   1:  PR[91,1] = PR[90,1] + 65.061;
   1:  PR[91,2] = PR[90,2] + 20.209;
   1:  PR[91,3] = PR[90,3] + 40.021;
   1:L PR[91] R[100]mm/sec CNT100;
   1:  PR[91,1] = PR[90,1] + 64.587;
   1:  PR[91,2] = PR[90,2] + 20.192;
   1:  PR[91,3] = PR[90,3] + 40.032;
   1:L PR[91] R[100]mm/sec CNT100;
   1:  PR[91,1] = PR[90,1] + 62.627;
   1:  PR[91,2] = PR[90,2] + 19.900;
   1:  PR[91,3] = PR[90,3] + 40.034;
   1:L PR[91] R[100]mm/sec CNT100;
   1:  PR[91,1] = PR[90,1] + 59.327;
   1:  PR[91,2] = PR[90,2] + 19.529;
   1:  PR[91,3] = PR[90,3] + 40.039;
   1:L PR[91] R[100]mm/sec CNT100;
   1:  PR[91,1] = PR[90,1] + 58.031;
   1:  PR[91,2] = PR[90,2] + 19.249;
   1:  PR[91,3] = PR[90,3] + 40.048;
   1:L PR[91] R[100]mm/sec CNT100;
   1:  PR[91,1] = PR[90,1] + 54.681;
   1:  PR[91,2] = PR[90,2] + 18.124;
   1:  PR[91,3] = PR[90,3] + 40.052;
   1:L PR[91] R[100]mm/sec CNT100;
   1:  PR[91,1] = PR[90,1] + 51.281;
   1:  PR[91,2] = PR[90,2] + 16.624;
   1:  PR[91,3] = PR[90,3] + 40.061;
   1:L PR[91] R[100]mm/sec CNT100;
   1:  PR[91,1] = PR[90,1] + 50.557;
   1:  PR[91,2] = PR[90,2] + 16.178;
   1:  PR[91,3] = PR[90,3] + 40.071;
   1:L PR[91] R[100]mm/sec CNT100;
   1:  PR[91,1] = PR[90,1] + 48.787;
   1:  PR[91,2] = PR[90,2] + 14.870;
   1:  PR[91,3] = PR[90,3] + 40.074;
   1:L PR[91] R[100]mm/sec CNT100;
   1:  PR[91,1] = PR[90,1] + 46.675;
   1:  PR[91,2] = PR[90,2] + 13.473;
   1:  PR[91,3] = PR[90,3] + 40.080;
   1:L PR[91] R[100]mm/sec CNT100;
   1:  PR[91,1] = PR[90,1] + 45.788;
   1:  PR[91,2] = PR[90,2] + 12.843;
   1:  PR[91,3] = PR[90,3] + 40.086;
   1:L PR[91] R[100]mm/sec CNT100;
   1:  PR[91,1] = PR[90,1] + 42.110;
   1:  PR[91,2] = PR[90,2] + 8.950;
   1:  PR[91,3] = PR[90,3] + 40.089;
   1:L PR[91] R[100]mm/sec CNT100;
   1:  PR[91,1] = PR[90,1] + 38.518;
   1:  PR[91,2] = PR[90,2] + 13.534;
   1:  PR[91,3] = PR[90,3] + 40.104;
   1:L PR[91] R[100]mm/sec CNT100;
   1:  PR[91,1] = PR[90,1] + 37.865;
   1:  PR[91,2] = PR[90,2] + 14.181;
   1:  PR[91,3] = PR[90,3] + 40.120;
